KUKA KRL program: EPS_2_251349_CBMH082_A_20251001124258.src

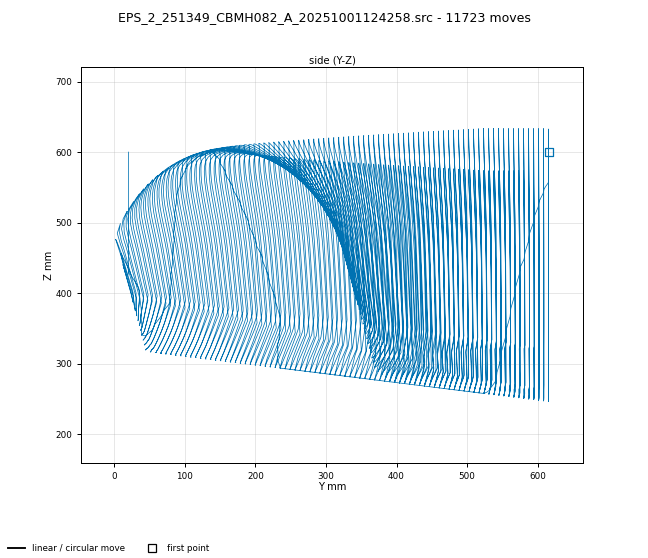
[picture p0: tool path of EPS_2_251349_CBMH082_A_20251001124258.src, 11723 of 11725 moves have a stored position in this frame; points joined in program order, loops and branches not executed]
&ACCESS RVP
&REL 4
&COMMENT QRS 19112012
&PARAM EDITMASK = *
DEF PART()
EXT BAS (BAS_COMMAND :IN,REAL :IN )
INT I
BAS (#INITMOV,0 )

;KUKA QRS Post kuka4.cps  Date:22-06-2017 !

File_ID=2859

QRS_PRE_INIT()

;Init var - Until changes are made in qrs_pre_init
Outlet_Square_prg=0
Inlet_1_Square_prg=0
Inlet_2_Square_prg=0
Inlet_3_Square_prg=0
Inlet_4_Square_prg=0
Inlet_5_Square_prg=0

Outlet_1={X 0.000, Y 523.550, Z 484.000, B 0.000, E1 0.000 }
Inlet_1={X 0.000, Y 527.930, Z 424.000, B 0.000, E1 90.000 }
Outlet_1_type=299
Inlet_1_type=299
;QRS#1=Sidecore dimensions
;QRS#2=300-12" PVC SDR 35
;QRS#3=300-12" PVC SDR 35
;QRS#4=
;QRS#5=
;QRS#6=
;QRS#7=
;QRS#8=
;QRS#9=16M PSX
;QRS#10=16M PSX
;QRS#11=
;QRS#12=
;QRS#13=
;QRS#14=
;QRS#15=
;QRS#16=1220x127x914 3'
;QRS#17=EPS Height
;QRS#18=633,5
;QRS#19=*
;QRS#20= UPDATED VERSION 22-06-2017
;QRS#21=*
Outlet_Square=0150
Inlet_1_Square=0150
Inlet_2_Square=0
Inlet_3_Square=0
Inlet_4_Square=0
Inlet_5_Square=0
Mill_Square=1
Outlet_Square_Prg=206
Inlet_1_Square_prg=206

QRS_INIT()

$ADVANCE=5

; T1
PTP {E1 173.526,E2 173.526}
PTP {X 0,Y 615.503,A -85,B 0,C 180,E1 173.526,E2 173.526,E3 0,E4 0,E5 0,E6 0}
QRS_SPEED_INIT()
LIN {X 0,Y 615.503,Z 600,A -85,B 0,C 180,E1 173.526,E2 173.526,E3 0,E4 0,E5 0,E6 0} C_VEL
LIN {X 0,Y 615.503,Z 569.829,A -85,B 0,C 180,E1 173.526,E2 173.526} C_VEL
LIN {X 0,Y 615.503,Z 560.181,A -85,B 0,C 180,E1 173.526,E2 173.526} C_VEL
LIN {X 0,Y 615.497,Z 558.359,A -85,B 0,C 180,E1 173.417,E2 173.417} C_VEL
LIN {X 0,Y 615.491,Z 551.664,A -85,B 0,C 180,E1 172.125,E2 172.125} C_VEL
LIN {X 0,Y 615.491,Z 543.149,A -85,B 0,C 180,E1 170.802,E2 170.802} C_VEL
LIN {X 0,Y 615.497,Z 534.071,A -85,B 0,C 180,E1 169.64,E2 169.64} C_VEL
LIN {X 0,Y 615.492,Z 524.798,A -85,B 0,C 180,E1 168.641,E2 168.641} C_VEL
LIN {X 0,Y 615.497,Z 512.83,A -85,B 0,C 180,E1 167.554,E2 167.554} C_VEL
LIN {X 0,Y 615.497,Z 500.591,A -85,B 0,C 180,E1 166.632,E2 166.632} C_VEL
LIN {X 0,Y 615.499,Z 487.891,A -85,B 0,C 180,E1 165.835,E2 165.835} C_VEL
LIN {X 0,Y 615.49,Z 473.795,A -85,B 0,C 180,E1 165.113,E2 165.113} C_VEL
LIN {X 0,Y 615.495,Z 459.141,A -85,B 0,C 180,E1 164.52,E2 164.52} C_VEL
LIN {X 0,Y 615.491,Z 444.202,A -85,B 0,C 180,E1 164.063,E2 164.063} C_VEL
LIN {X 0,Y 615.486,Z 428.985,A -85,B 0,C 180,E1 163.738,E2 163.738} C_VEL
LIN {X 0,Y 615.463,Z 380.474,A -85,B 0,C 180,E1 163.136,E2 163.136} C_VEL
LIN {X 0,Y 615.477,Z 263.406,A -85,B 0,C 180,E1 161.724,E2 161.724} C_VEL
LIN {X 0,Y 615.454,Z 246.316,A -85,B 0,C 180,E1 159.315,E2 159.315} C_VEL
LIN {X 0,Y 615.493,Z 246.313,A -85,B 0,C 180,E1 156.445,E2 156.445} C_VEL
LIN {X 0,Y 615.457,Z 246.319,A -85,B 0,C 180,E1 153.555,E2 153.555} C_VEL
LIN {X 0,Y 615.454,Z 246.316,A -85,B 0,C 180,E1 151.341,E2 151.341} C_VEL
LIN {X 0,Y 615.474,Z 246.311,A -85,B 0,C 180,E1 148.917,E2 148.917} C_VEL
LIN {X 0,Y 615.481,Z 246.324,A -85,B 0,C 180,E1 145.979,E2 145.979} C_VEL
LIN {X 0,Y 615.456,Z 246.318,A -85,B 0,C 180,E1 143.574,E2 143.574} C_VEL
LIN {X 0,Y 615.473,Z 246.311,A -85,B 0,C 180,E1 140.94,E2 140.94} C_VEL
LIN {X 0,Y 615.474,Z 246.322,A -85,B 0,C 180,E1 137.922,E2 137.922} C_VEL
LIN {X 0,Y 615.467,Z 246.321,A -85,B 0,C 180,E1 135.85,E2 135.85} C_VEL
LIN {X 0,Y 615.458,Z 246.314,A -85,B 0,C 180,E1 133.248,E2 133.248} C_VEL
LIN {X 0,Y 615.488,Z 246.314,A -85,B 0,C 180,E1 130.607,E2 130.607} C_VEL
LIN {X 0,Y 615.477,Z 246.323,A -85,B 0,C 180,E1 128.012,E2 128.012} C_VEL
LIN {X 0,Y 615.453,Z 246.318,A -85,B 0,C 180,E1 125.619,E2 125.619} C_VEL
LIN {X 0,Y 615.461,Z 246.313,A -85,B 0,C 180,E1 123.239,E2 123.239} C_VEL
LIN {X 0,Y 615.489,Z 246.309,A -85,B 0,C 180,E1 120.92,E2 120.92} C_VEL
LIN {X 0,Y 615.464,Z 246.321,A -85,B 0,C 180,E1 117.917,E2 117.917} C_VEL
LIN {X 0,Y 615.452,Z 246.317,A -85,B 0,C 180,E1 115.564,E2 115.564} C_VEL
LIN {X 0,Y 615.487,Z 246.312,A -85,B 0,C 180,E1 112.845,E2 112.845} C_VEL
LIN {X 0,Y 615.469,Z 246.322,A -85,B 0,C 180,E1 110.034,E2 110.034} C_VEL
LIN {X 0,Y 615.463,Z 246.321,A -85,B 0,C 180,E1 107.958,E2 107.958} C_VEL
LIN {X 0,Y 615.459,Z 246.32,A -85,B 0,C 180,E1 105.907,E2 105.907} C_VEL
LIN {X 0,Y 615.457,Z 246.319,A -85,B 0,C 180,E1 103.876,E2 103.876} C_VEL
LIN {X 0,Y 615.472,Z 246.311,A -85,B 0,C 180,E1 101.194,E2 101.194} C_VEL
LIN {X 0,Y 615.491,Z 246.322,A -85,B 0,C 180,E1 98.537,E2 98.537} C_VEL
LIN {X 0,Y 615.456,Z 246.319,A -85,B 0,C 180,E1 95.9,E2 95.9} C_VEL
LIN {X 0,Y 615.469,Z 246.312,A -85,B 0,C 180,E1 93.274,E2 93.274} C_VEL
LIN {X 0,Y 615.493,Z 246.319,A -85,B 0,C 180,E1 90.655,E2 90.655} C_VEL
LIN {X 0,Y 615.461,Z 246.32,A -85,B 0,C 180,E1 88.038,E2 88.038} C_VEL
LIN {X 0,Y 615.461,Z 246.313,A -85,B 0,C 180,E1 85.416,E2 85.416} C_VEL
LIN {X 0,Y 615.493,Z 246.316,A -85,B 0,C 180,E1 82.785,E2 82.785} C_VEL
LIN {X 0,Y 615.464,Z 246.321,A -85,B 0,C 180,E1 80.138,E2 80.138} C_VEL
LIN {X 0,Y 615.461,Z 246.313,A -85,B 0,C 180,E1 77.47,E2 77.47} C_VEL
LIN {X 0,Y 615.493,Z 246.318,A -85,B 0,C 180,E1 74.775,E2 74.775} C_VEL
LIN {X 0,Y 615.456,Z 246.319,A -85,B 0,C 180,E1 72.043,E2 72.043} C_VEL
LIN {X 0,Y 615.466,Z 246.312,A -85,B 0,C 180,E1 69.446,E2 69.446} C_VEL
LIN {X 0,Y 615.485,Z 246.311,A -85,B 0,C 180,E1 67.157,E2 67.157} C_VEL
LIN {X 0,Y 615.464,Z 246.322,A -85,B 0,C 180,E1 64.285,E2 64.285} C_VEL
LIN {X 0,Y 615.454,Z 246.319,A -85,B 0,C 180,E1 62.085,E2 62.085} C_VEL
LIN {X 0,Y 615.449,Z 246.317,A -85,B 0,C 180,E1 59.839,E2 59.839} C_VEL
LIN {X 0,Y 615.464,Z 246.313,A -85,B 0,C 180,E1 57.543,E2 57.543} C_VEL
LIN {X 0,Y 615.499,Z 246.309,A -85,B 0,C 180,E1 55.187,E2 55.187} C_VEL
LIN {X 0,Y 615.488,Z 246.324,A -85,B 0,C 180,E1 52.759,E2 52.759} C_VEL
LIN {X 0,Y 615.459,Z 246.32,A -85,B 0,C 180,E1 50.249,E2 50.249} C_VEL
LIN {X 0,Y 615.457,Z 246.314,A -85,B 0,C 180,E1 47.646,E2 47.646} C_VEL
LIN {X 0,Y 615.489,Z 246.319,A -85,B 0,C 180,E1 44.933,E2 44.933} C_VEL
LIN {X 0,Y 615.463,Z 246.321,A -85,B 0,C 180,E1 42.354,E2 42.354} C_VEL
LIN {X 0,Y 615.457,Z 246.314,A -85,B 0,C 180,E1 39.751,E2 39.751} C_VEL
LIN {X 0,Y 615.486,Z 246.322,A -85,B 0,C 180,E1 36.939,E2 36.939} C_VEL
LIN {X 0,Y 615.448,Z 246.317,A -85,B 0,C 180,E1 34.023,E2 34.023} C_VEL
LIN {X 0,Y 615.494,Z 246.316,A -85,B 0,C 180,E1 31.09,E2 31.09} C_VEL
LIN {X 0,Y 615.463,Z 246.321,A -85,B 0,C 180,E1 28.449,E2 28.449} C_VEL
LIN {X 0,Y 615.462,Z 246.321,A -85,B 0,C 180,E1 26.444,E2 26.444} C_VEL
LIN {X 0,Y 615.449,Z 246.316,A -85,B 0,C 180,E1 24.004,E2 24.004} C_VEL
LIN {X 0,Y 615.492,Z 246.31,A -85,B 0,C 180,E1 21.431,E2 21.431} C_VEL
LIN {X 0,Y 615.47,Z 246.322,A -85,B 0,C 180,E1 18.604,E2 18.604} C_VEL
LIN {X 0,Y 615.457,Z 246.32,A -85,B 0,C 180,E1 16.427,E2 16.427} C_VEL
LIN {X 0,Y 615.458,Z 246.314,A -85,B 0,C 180,E1 13.874,E2 13.874} C_VEL
LIN {X 0,Y 615.485,Z 246.328,A -85,B 0,C 180,E1 10.895,E2 10.895} C_VEL
LIN {X 0,Y 615.461,Z 246.321,A -85,B 0,C 180,E1 8.536,E2 8.536} C_VEL
LIN {X 0,Y 615.459,Z 246.314,A -85,B 0,C 180,E1 5.898,E2 5.898} C_VEL
LIN {X 0,Y 615.494,Z 246.316,A -85,B 0,C 180,E1 3.272,E2 3.272} C_VEL
LIN {X 0,Y 615.466,Z 246.322,A -85,B 0,C 180,E1 0.654,E2 0.654} C_VEL
LIN {X 0,Y 615.454,Z 246.315,A -85,B 0,C 180,E1 -1.964,E2 -1.964} C_VEL
LIN {X 0,Y 615.496,Z 246.313,A -85,B 0,C 180,E1 -4.585,E2 -4.585} C_VEL
LIN {X 0,Y 615.473,Z 246.322,A -85,B 0,C 180,E1 -7.216,E2 -7.216} C_VEL
LIN {X 0,Y 615.45,Z 246.316,A -85,B 0,C 180,E1 -9.863,E2 -9.863} C_VEL
LIN {X 0,Y 615.49,Z 246.314,A -85,B 0,C 180,E1 -12.53,E2 -12.53} C_VEL
LIN {X 0,Y 615.468,Z 246.322,A -85,B 0,C 180,E1 -15.227,E2 -15.227} C_VEL
LIN {X 0,Y 615.463,Z 246.321,A -85,B 0,C 180,E1 -17.272,E2 -17.272} C_VEL
LIN {X 0,Y 615.454,Z 246.321,A -85,B 0,C 180,E1 -19.339,E2 -19.339} C_VEL
LIN {X 0,Y 615.453,Z 246.319,A -85,B 0,C 180,E1 -21.433,E2 -21.433} C_VEL
LIN {X 0,Y 615.459,Z 246.314,A -85,B 0,C 180,E1 -24.006,E2 -24.006} C_VEL
LIN {X 0,Y 615.497,Z 246.312,A -85,B 0,C 180,E1 -26.444,E2 -26.444} C_VEL
LIN {X 0,Y 615.494,Z 246.319,A -85,B 0,C 180,E1 -28.658,E2 -28.658} C_VEL
LIN {X 0,Y 615.471,Z 246.322,A -85,B 0,C 180,E1 -31.086,E2 -31.086} C_VEL
LIN {X 0,Y 615.449,Z 246.318,A -85,B 0,C 180,E1 -33.531,E2 -33.531} C_VEL
LIN {X 0,Y 615.455,Z 246.314,A -85,B 0,C 180,E1 -35.832,E2 -35.832} C_VEL
LIN {X 0,Y 615.475,Z 246.312,A -85,B 0,C 180,E1 -38.07,E2 -38.07} C_VEL
LIN {X 0,Y 615.466,Z 246.322,A -85,B 0,C 180,E1 -41.094,E2 -41.094} C_VEL
LIN {X 0,Y 615.455,Z 246.32,A -85,B 0,C 180,E1 -43.248,E2 -43.248} C_VEL
LIN {X 0,Y 615.472,Z 246.312,A -85,B 0,C 180,E1 -46.004,E2 -46.004} C_VEL
LIN {X 0,Y 615.476,Z 246.324,A -85,B 0,C 180,E1 -48.907,E2 -48.907} C_VEL
LIN {X 0,Y 615.461,Z 246.321,A -85,B 0,C 180,E1 -51.095,E2 -51.095} C_VEL
LIN {X 0,Y 615.45,Z 246.316,A -85,B 0,C 180,E1 -53.574,E2 -53.574} C_VEL
LIN {X 0,Y 615.494,Z 246.318,A -85,B 0,C 180,E1 -56.465,E2 -56.465} C_VEL
LIN {X 0,Y 615.457,Z 246.321,A -85,B 0,C 180,E1 -59.08,E2 -59.08} C_VEL
LIN {X 0,Y 615.45,Z 246.316,A -85,B 0,C 180,E1 -61.556,E2 -61.556} C_VEL
LIN {X 0,Y 615.462,Z 246.374,A -85,B 0,C 180,E1 -63.784,E2 -63.784} C_VEL
LIN {X 0,Y 615.485,Z 272.614,A -85,B 0,C 180,E1 -66.623,E2 -66.623} C_VEL
LIN {X 0,Y 615.486,Z 299.254,A -85,B 0,C 180,E1 -69.443,E2 -69.443} C_VEL
LIN {X 0,Y 615.495,Z 321.324,A -85,B 0,C 180,E1 -71.741,E2 -71.741} C_VEL
LIN {X 0,Y 615.487,Z 488.149,A -85,B 0,C 180,E1 -73.768,E2 -73.768} C_VEL
LIN {X 0,Y 615.49,Z 503.756,A -85,B 0,C 180,E1 -74.096,E2 -74.096} C_VEL
LIN {X 0,Y 615.48,Z 519.082,A -85,B 0,C 180,E1 -74.563,E2 -74.563} C_VEL
LIN {X 0,Y 615.492,Z 532.779,A -85,B 0,C 180,E1 -75.114,E2 -75.114} C_VEL
LIN {X 0,Y 615.494,Z 547.055,A -85,B 0,C 180,E1 -75.834,E2 -75.834} C_VEL
LIN {X 0,Y 615.497,Z 559.915,A -85,B 0,C 180,E1 -76.632,E2 -76.632} C_VEL
LIN {X 0,Y 615.495,Z 572.268,A -85,B 0,C 180,E1 -77.555,E2 -77.555} C_VEL
LIN {X 0,Y 615.495,Z 582.618,A -85,B 0,C 180,E1 -78.474,E2 -78.474} C_VEL
LIN {X 0,Y 615.495,Z 592.193,A -85,B 0,C 180,E1 -79.474,E2 -79.474} C_VEL
LIN {X 0,Y 615.494,Z 601.585,A -85,B 0,C 180,E1 -80.637,E2 -80.637} C_VEL
LIN {X 0,Y 615.495,Z 609.387,A -85,B 0,C 180,E1 -81.795,E2 -81.795} C_VEL
LIN {X 0,Y 615.496,Z 616.609,A -85,B 0,C 180,E1 -83.102,E2 -83.102} C_VEL
LIN {X 0,Y 615.499,Z 622.44,A -85,B 0,C 180,E1 -84.431,E2 -84.431} C_VEL
LIN {X 0,Y 615.491,Z 625.863,A -85,B 0,C 180,E1 -85.416,E2 -85.416} C_VEL
LIN {X 0,Y 615.492,Z 629.32,A -85,B 0,C 180,E1 -86.728,E2 -86.728} C_VEL
LIN {X 0,Y 615.497,Z 631.594,A -85,B 0,C 180,E1 -88.038,E2 -88.038} C_VEL
LIN {X 0,Y 615.493,Z 632.741,A -85,B 0,C 180,E1 -89.347,E2 -89.347} C_VEL
LIN {X 0,Y 615.493,Z 632.74,A -85,B 0,C 180,E1 -90.655,E2 -90.655} C_VEL
LIN {X 0,Y 615.497,Z 631.592,A -85,B 0,C 180,E1 -91.964,E2 -91.964} C_VEL
LIN {X 0,Y 615.492,Z 629.316,A -85,B 0,C 180,E1 -93.274,E2 -93.274} C_VEL
LIN {X 0,Y 615.491,Z 625.857,A -85,B 0,C 180,E1 -94.585,E2 -94.585} C_VEL
LIN {X 0,Y 615.49,Z 621.14,A -85,B 0,C 180,E1 -95.899,E2 -95.899} C_VEL
LIN {X 0,Y 615.495,Z 615.025,A -85,B 0,C 180,E1 -97.216,E2 -97.216} C_VEL
LIN {X 0,Y 615.49,Z 607.327,A -85,B 0,C 180,E1 -98.537,E2 -98.537} C_VEL
LIN {X 0,Y 615.495,Z 599.107,A -85,B 0,C 180,E1 -99.697,E2 -99.697} C_VEL
LIN {X 0,Y 615.497,Z 588.896,A -85,B 0,C 180,E1 -100.892,E2 -100.892} C_VEL
LIN {X 0,Y 615.495,Z 579.059,A -85,B 0,C 180,E1 -101.861,E2 -101.861} C_VEL
LIN {X 0,Y 615.498,Z 566.936,A -85,B 0,C 180,E1 -102.866,E2 -102.866} C_VEL
LIN {X 0,Y 615.498,Z 554.785,A -85,B 0,C 180,E1 -103.706,E2 -103.706} C_VEL
LIN {X 0,Y 615.484,Z 541.367,A -85,B 0,C 180,E1 -104.473,E2 -104.473} C_VEL
LIN {X 0,Y 615.495,Z 526.83,A -85,B 0,C 180,E1 -105.142,E2 -105.142} C_VEL
LIN {X 0,Y 615.484,Z 512.592,A -85,B 0,C 180,E1 -105.651,E2 -105.651} C_VEL
LIN {X 0,Y 615.499,Z 498.103,A -85,B 0,C 180,E1 -106.036,E2 -106.036} C_VEL
LIN {X 0,Y 615.487,Z 483.529,A -85,B 0,C 180,E1 -106.298,E2 -106.298} C_VEL
LIN {X 0,Y 615.494,Z 321.314,A -85,B 0,C 180,E1 -108.26,E2 -108.26} C_VEL
LIN {X 0,Y 615.484,Z 295.921,A -85,B 0,C 180,E1 -110.907,E2 -110.907} C_VEL
LIN {X 0,Y 615.491,Z 268.818,A -85,B 0,C 180,E1 -113.783,E2 -113.783} C_VEL
LIN {X 0,Y 615.463,Z 246.356,A -85,B 0,C 180,E1 -116.218,E2 -116.218} C_VEL
LIN {X 0,Y 615.455,Z 246.318,A -85,B 0,C 180,E1 -118.66,E2 -118.66} C_VEL
LIN {X 0,Y 615.485,Z 246.324,A -85,B 0,C 180,E1 -121.085,E2 -121.085} C_VEL
LIN {X 0,Y 615.478,Z 246.31,A -85,B 0,C 180,E1 -124.023,E2 -124.023} C_VEL
LIN {X 0,Y 615.464,Z 246.316,A -85,B 0,C 180,E1 -126.427,E2 -126.427} C_VEL
LIN {X 0,Y 615.493,Z 246.324,A -85,B 0,C 180,E1 -129.063,E2 -129.063} C_VEL
LIN {X 0,Y 615.484,Z 246.313,A -85,B 0,C 180,E1 -131.475,E2 -131.475} C_VEL
LIN {X 0,Y 615.475,Z 246.313,A -85,B 0,C 180,E1 -134.151,E2 -134.151} C_VEL
LIN {X 0,Y 615.486,Z 246.321,A -85,B 0,C 180,E1 -136.953,E2 -136.953} C_VEL
LIN {X 0,Y 615.479,Z 246.312,A -85,B 0,C 180,E1 -139.393,E2 -139.393} C_VEL
LIN {X 0,Y 615.484,Z 246.311,A -85,B 0,C 180,E1 -141.989,E2 -141.989} C_VEL
LIN {X 0,Y 615.489,Z 246.321,A -85,B 0,C 180,E1 -144.384,E2 -144.384} C_VEL
LIN {X 0,Y 615.476,Z 246.321,A -85,B 0,C 180,E1 -146.763,E2 -146.763} C_VEL
LIN {X 0,Y 615.465,Z 246.315,A -85,B 0,C 180,E1 -149.079,E2 -149.079} C_VEL
LIN {X 0,Y 615.489,Z 246.308,A -85,B 0,C 180,E1 -151.55,E2 -151.55} C_VEL
LIN {X 0,Y 615.483,Z 246.323,A -85,B 0,C 180,E1 -154.433,E2 -154.433} C_VEL
LIN {X 0,Y 615.46,Z 246.314,A -85,B 0,C 180,E1 -157.154,E2 -157.154} C_VEL
LIN {X 0,Y 615.48,Z 246.437,A -85,B 0,C 180,E1 -159.446,E2 -159.446} C_VEL
LIN {X 0,Y 615.494,Z 263.458,A -85,B 0,C 180,E1 -161.822,E2 -161.822} C_VEL
LIN {X 0,Y 615.497,Z 427.262,A -85,B 0,C 180,E1 -163.8,E2 -163.8} C_VEL
LIN {X 0,Y 615.494,Z 441.803,A -85,B 0,C 180,E1 -164.095,E2 -164.095} C_VEL
LIN {X 0,Y 615.496,Z 456.406,A -85,B 0,C 180,E1 -164.519,E2 -164.519} C_VEL
LIN {X 0,Y 615.489,Z 469.73,A -85,B 0,C 180,E1 -165.028,E2 -165.028} C_VEL
LIN {X 0,Y 615.493,Z 483.381,A -85,B 0,C 180,E1 -165.681,E2 -165.681} C_VEL
LIN {X 0,Y 615.5,Z 496.661,A -85,B 0,C 180,E1 -166.462,E2 -166.462} C_VEL
LIN {X 0,Y 615.497,Z 508.512,A -85,B 0,C 180,E1 -167.302,E2 -167.302} C_VEL
LIN {X 0,Y 615.497,Z 520.356,A -85,B 0,C 180,E1 -168.306,E2 -168.306} C_VEL
LIN {X 0,Y 615.495,Z 530.169,A -85,B 0,C 180,E1 -169.292,E2 -169.292} C_VEL
LIN {X 0,Y 615.498,Z 540.009,A -85,B 0,C 180,E1 -170.469,E2 -170.469} C_VEL
LIN {X 0,Y 615.496,Z 548.1,A -85,B 0,C 180,E1 -171.628,E2 -171.628} C_VEL
LIN {X 0,Y 615.493,Z 554.78,A -85,B 0,C 180,E1 -172.784,E2 -172.784} C_VEL
LIN {X 0,Y 615.488,Z 560.948,A -85,B 0,C 180,E1 -174.101,E2 -174.101} C_VEL
LIN {X 0,Y 615.489,Z 565.715,A -85,B 0,C 180,E1 -175.415,E2 -175.415} C_VEL
LIN {X 0,Y 615.496,Z 569.219,A -85,B 0,C 180,E1 -176.727,E2 -176.727} C_VEL
LIN {X 0,Y 615.493,Z 571.541,A -85,B 0,C 180,E1 -178.036,E2 -178.036} C_VEL
LIN {X 0,Y 615.491,Z 572.728,A -85,B 0,C 180,E1 -179.345,E2 -179.345} C_VEL
LIN {X 0,Y 615.494,Z 572.751,A -85,B 0,C 180,E1 -180.654,E2 -180.654} C_VEL
LIN {X 0,Y 615.497,Z 571.647,A -85,B 0,C 180,E1 -181.963,E2 -181.963} C_VEL
LIN {X 0,Y 615.497,Z 569.416,A -85,B 0,C 180,E1 -183.272,E2 -183.272} C_VEL
LIN {X 0,Y 615.496,Z 566.005,A -85,B 0,C 180,E1 -184.584,E2 -184.584} C_VEL
LIN {X 0,Y 615.49,Z 561.34,A -85,B 0,C 180,E1 -185.898,E2 -185.898} C_VEL
LIN {X 0,Y 615.497,Z 558.359,A -85,B 0,C 180,E1 -186.583,E2 -186.583} C_VEL
LIN {X 0,Y 614.828,Z 556.102,A -85,B 0,C 180,E1 -187.082,E2 -187.082} C_VEL
LIN {X 0,Y 612.006,Z 552.209,A -85,B 0,C 180,E1 -187.888,E2 -187.888} C_VEL
LIN {X 0,Y 609.154,Z 547.637,A -85,B 0,C 180,E1 -188.679,E2 -188.679} C_VEL
LIN {X 0,Y 608.464,Z 544.491,A -85,B 0,C 180,E1 -189.153,E2 -189.153} C_VEL
LIN {X 0,Y 608.478,Z 535.67,A -85,B 0,C 180,E1 -190.312,E2 -190.312} C_VEL
LIN {X 0,Y 608.494,Z 524.953,A -85,B 0,C 180,E1 -191.492,E2 -191.492} C_VEL
LIN {X 0,Y 608.513,Z 512.908,A -85,B 0,C 180,E1 -192.591,E2 -192.591} C_VEL
LIN {X 0,Y 608.543,Z 500.629,A -85,B 0,C 180,E1 -193.524,E2 -193.524} C_VEL
LIN {X 0,Y 608.577,Z 487.683,A -85,B 0,C 180,E1 -194.341,E2 -194.341} C_VEL
LIN {X 0,Y 608.605,Z 473.771,A -85,B 0,C 180,E1 -195.059,E2 -195.059} C_VEL
LIN {X 0,Y 608.639,Z 459.125,A -85,B 0,C 180,E1 -195.658,E2 -195.658} C_VEL
LIN {X 0,Y 608.661,Z 443.559,A -85,B 0,C 180,E1 -196.137,E2 -196.137} C_VEL
LIN {X 0,Y 608.678,Z 427.766,A -85,B 0,C 180,E1 -196.469,E2 -196.469} C_VEL
LIN {X 0,Y 608.638,Z 264.297,A -85,B 0,C 180,E1 -198.468,E2 -198.468} C_VEL
LIN {X 0,Y 608.509,Z 263.438,A -85,B 0,C 180,E1 -198.492,E2 -198.492} C_VEL
LIN {X 0,Y 608.466,Z 247.558,A -85,B 0,C 180,E1 -200.735,E2 -200.735} C_VEL
LIN {X 0,Y 608.444,Z 247.315,A -85,B 0,C 180,E1 -200.981,E2 -200.981} C_VEL
LIN {X 0,Y 608.469,Z 247.319,A -85,B 0,C 180,E1 -203.844,E2 -203.844} C_VEL
LIN {X 0,Y 608.437,Z 247.323,A -85,B 0,C 180,E1 -206.035,E2 -206.035} C_VEL
LIN {X 0,Y 608.447,Z 247.314,A -85,B 0,C 180,E1 -208.615,E2 -208.615} C_VEL
LIN {X 0,Y 608.445,Z 247.315,A -85,B 0,C 180,E1 -211.317,E2 -211.317} C_VEL
LIN {X 0,Y 608.475,Z 247.317,A -85,B 0,C 180,E1 -213.735,E2 -213.735} C_VEL
LIN {X 0,Y 608.442,Z 247.32,A -85,B 0,C 180,E1 -216.091,E2 -216.091} C_VEL
LIN {X 0,Y 608.424,Z 247.316,A -85,B 0,C 180,E1 -218.59,E2 -218.59} C_VEL
LIN {X 0,Y 608.461,Z 247.314,A -85,B 0,C 180,E1 -221.341,E2 -221.341} C_VEL
LIN {X 0,Y 608.465,Z 247.321,A -85,B 0,C 180,E1 -223.869,E2 -223.869} C_VEL
LIN {X 0,Y 608.449,Z 247.313,A -85,B 0,C 180,E1 -226.692,E2 -226.692} C_VEL
LIN {X 0,Y 608.434,Z 247.314,A -85,B 0,C 180,E1 -228.821,E2 -228.821} C_VEL
LIN {X 0,Y 608.464,Z 247.322,A -85,B 0,C 180,E1 -231.759,E2 -231.759} C_VEL
LIN {X 0,Y 608.439,Z 247.321,A -85,B 0,C 180,E1 -233.954,E2 -233.954} C_VEL
LIN {X 0,Y 608.437,Z 247.316,A -85,B 0,C 180,E1 -236.327,E2 -236.327} C_VEL
LIN {X 0,Y 608.437,Z 247.314,A -85,B 0,C 180,E1 -238.732,E2 -238.732} C_VEL
LIN {X 0,Y 608.478,Z 247.314,A -85,B 0,C 180,E1 -241.377,E2 -241.377} C_VEL
LIN {X 0,Y 608.444,Z 247.315,A -85,B 0,C 180,E1 -244.282,E2 -244.282} C_VEL
LIN {X 0,Y 608.439,Z 247.314,A -85,B 0,C 180,E1 -246.875,E2 -246.875} C_VEL
LIN {X 0,Y 608.457,Z 247.322,A -85,B 0,C 180,E1 -249.725,E2 -249.725} C_VEL
LIN {X 0,Y 608.435,Z 247.322,A -85,B 0,C 180,E1 -251.827,E2 -251.827} C_VEL
LIN {X 0,Y 608.448,Z 247.319,A -85,B 0,C 180,E1 -253.905,E2 -253.905} C_VEL
LIN {X 0,Y 608.445,Z 247.318,A -85,B 0,C 180,E1 -255.988,E2 -255.988} C_VEL
LIN {X 0,Y 608.446,Z 247.313,A -85,B 0,C 180,E1 -258.675,E2 -258.675} C_VEL
LIN {X 0,Y 608.457,Z 247.318,A -85,B 0,C 180,E1 -261.363,E2 -261.363} C_VEL
LIN {X 0,Y 608.435,Z 247.318,A -85,B 0,C 180,E1 -264.032,E2 -264.032} C_VEL
LIN {X 0,Y 608.462,Z 247.311,A -85,B 0,C 180,E1 -266.688,E2 -266.688} C_VEL
LIN {X 0,Y 608.486,Z 247.315,A -85,B 0,C 180,E1 -269.337,E2 -269.337} C_VEL
LIN {X 0,Y 608.431,Z 247.318,A -85,B 0,C 180,E1 -271.985,E2 -271.985} C_VEL
LIN {X 0,Y 608.43,Z 247.318,A -85,B 0,C 180,E1 -273.973,E2 -273.973} C_VEL
LIN {X 0,Y 608.449,Z 247.313,A -85,B 0,C 180,E1 -276.632,E2 -276.632} C_VEL
LIN {X 0,Y 608.469,Z 247.317,A -85,B 0,C 180,E1 -279.305,E2 -279.305} C_VEL
LIN {X 0,Y 608.44,Z 247.316,A -85,B 0,C 180,E1 -281.999,E2 -281.999} C_VEL
LIN {X 0,Y 608.461,Z 247.312,A -85,B 0,C 180,E1 -284.72,E2 -284.72} C_VEL
LIN {X 0,Y 608.448,Z 247.324,A -85,B 0,C 180,E1 -287.476,E2 -287.476} C_VEL
LIN {X 0,Y 608.437,Z 247.314,A -85,B 0,C 180,E1 -290.274,E2 -290.274} C_VEL
LIN {X 0,Y 608.445,Z 247.313,A -85,B 0,C 180,E1 -292.476,E2 -292.476} C_VEL
LIN {X 0,Y 608.449,Z 247.322,A -85,B 0,C 180,E1 -295.3,E2 -295.3} C_VEL
LIN {X 0,Y 608.437,Z 247.323,A -85,B 0,C 180,E1 -297.517,E2 -297.517} C_VEL
LIN {X 0,Y 608.438,Z 247.316,A -85,B 0,C 180,E1 -299.969,E2 -299.969} C_VEL
LIN {X 0,Y 608.441,Z 247.314,A -85,B 0,C 180,E1 -302.521,E2 -302.521} C_VEL
LIN {X 0,Y 608.44,Z 247.323,A -85,B 0,C 180,E1 -305.276,E2 -305.276} C_VEL
LIN {X 0,Y 608.447,Z 247.317,A -85,B 0,C 180,E1 -307.746,E2 -307.746} C_VEL
LIN {X 0,Y 608.427,Z 247.315,A -85,B 0,C 180,E1 -310.328,E2 -310.328} C_VEL
LIN {X 0,Y 608.455,Z 247.317,A -85,B 0,C 180,E1 -312.958,E2 -312.958} C_VEL
LIN {X 0,Y 608.427,Z 247.319,A -85,B 0,C 180,E1 -315.737,E2 -315.737} C_VEL
LIN {X 0,Y 608.432,Z 247.316,A -85,B 0,C 180,E1 -317.937,E2 -317.937} C_VEL
LIN {X 0,Y 608.467,Z 247.313,A -85,B 0,C 180,E1 -320.701,E2 -320.701} C_VEL
LIN {X 0,Y 608.455,Z 247.32,A -85,B 0,C 180,E1 -323.086,E2 -323.086} C_VEL
LIN {X 0,Y 608.458,Z 247.317,A -85,B 0,C 180,E1 -325.531,E2 -325.531} C_VEL
LIN {X 0,Y 608.441,Z 247.315,A -85,B 0,C 180,E1 -327.905,E2 -327.905} C_VEL
LIN {X 0,Y 608.443,Z 247.313,A -85,B 0,C 180,E1 -330.22,E2 -330.22} C_VEL
LIN {X 0,Y 608.479,Z 247.313,A -85,B 0,C 180,E1 -332.789,E2 -332.789} C_VEL
LIN {X 0,Y 608.437,Z 247.32,A -85,B 0,C 180,E1 -335.429,E2 -335.429} C_VEL
LIN {X 0,Y 608.458,Z 247.312,A -85,B 0,C 180,E1 -338.309,E2 -338.309} C_VEL
LIN {X 0,Y 608.456,Z 247.32,A -85,B 0,C 180,E1 -341.284,E2 -341.284} C_VEL
LIN {X 0,Y 608.431,Z 247.315,A -85,B 0,C 180,E1 -343.906,E2 -343.906} C_VEL
LIN {X 0,Y 608.462,Z 247.314,A -85,B 0,C 180,E1 -346.644,E2 -346.644} C_VEL
LIN {X 0,Y 608.448,Z 247.319,A -85,B 0,C 180,E1 -349.351,E2 -349.351} C_VEL
LIN {X 0,Y 608.453,Z 247.312,A -85,B 0,C 180,E1 -352.033,E2 -352.033} C_VEL
LIN {X 0,Y 608.469,Z 247.315,A -85,B 0,C 180,E1 -354.699,E2 -354.699} C_VEL
LIN {X 0,Y 608.457,Z 247.317,A -85,B 0,C 180,E1 -357.352,E2 -357.352} C_VEL
LIN {X 0,Y 608.448,Z 247.313,A -85,B 0,C 180,E1 -360.001,E2 -360.001} C_VEL
LIN {X 0,Y 608.483,Z 247.313,A -85,B 0,C 180,E1 -362.649,E2 -362.649} C_VEL
LIN {X 0,Y 608.449,Z 247.318,A -85,B 0,C 180,E1 -365.302,E2 -365.302} C_VEL
LIN {X 0,Y 608.451,Z 247.312,A -85,B 0,C 180,E1 -367.968,E2 -367.968} C_VEL
LIN {X 0,Y 608.468,Z 247.321,A -85,B 0,C 180,E1 -370.963,E2 -370.963} C_VEL
LIN {X 0,Y 608.442,Z 247.317,A -85,B 0,C 180,E1 -373.357,E2 -373.357} C_VEL
LIN {X 0,Y 608.45,Z 247.316,A -85,B 0,C 180,E1 -375.407,E2 -375.407} C_VEL
LIN {X 0,Y 608.429,Z 247.317,A -85,B 0,C 180,E1 -377.478,E2 -377.478} C_VEL
LIN {X 0,Y 608.425,Z 247.317,A -85,B 0,C 180,E1 -379.572,E2 -379.572} C_VEL
LIN {X 0,Y 608.443,Z 247.314,A -85,B 0,C 180,E1 -381.693,E2 -381.693} C_VEL
LIN {X 0,Y 608.449,Z 247.318,A -85,B 0,C 180,E1 -384.572,E2 -384.572} C_VEL
LIN {X 0,Y 608.428,Z 247.316,A -85,B 0,C 180,E1 -387.519,E2 -387.519} C_VEL
LIN {X 0,Y 608.444,Z 247.313,A -85,B 0,C 180,E1 -389.971,E2 -389.971} C_VEL
LIN {X 0,Y 608.447,Z 247.323,A -85,B 0,C 180,E1 -392.88,E2 -392.88} C_VEL
LIN {X 0,Y 608.426,Z 247.319,A -85,B 0,C 180,E1 -395.279,E2 -395.279} C_VEL
LIN {X 0,Y 608.45,Z 247.312,A -85,B 0,C 180,E1 -397.748,E2 -397.748} C_VEL
LIN {X 0,Y 608.448,Z 247.316,A -85,B 0,C 180,E1 -400.331,E2 -400.331} C_VEL
LIN {X 0,Y 608.439,Z 247.321,A -85,B 0,C 180,E1 -402.961,E2 -402.961} C_VEL
LIN {X 0,Y 608.432,Z 247.315,A -85,B 0,C 180,E1 -405.739,E2 -405.739} C_VEL
LIN {X 0,Y 608.446,Z 247.313,A -85,B 0,C 180,E1 -407.939,E2 -407.939} C_VEL
LIN {X 0,Y 608.469,Z 247.321,A -85,B 0,C 180,E1 -410.703,E2 -410.703} C_VEL
LIN {X 0,Y 608.432,Z 247.319,A -85,B 0,C 180,E1 -413.085,E2 -413.085} C_VEL
LIN {X 0,Y 608.443,Z 247.314,A -85,B 0,C 180,E1 -415.531,E2 -415.531} C_VEL
LIN {X 0,Y 608.448,Z 247.313,A -85,B 0,C 180,E1 -417.906,E2 -417.906} C_VEL
LIN {X 0,Y 608.482,Z 247.312,A -85,B 0,C 180,E1 -420.223,E2 -420.223} C_VEL
LIN {X 0,Y 608.422,Z 247.32,A -85,B 0,C 180,E1 -423.226,E2 -423.226} C_VEL
LIN {X 0,Y 608.437,Z 247.415,A -85,B 0,C 180,E1 -423.573,E2 -423.573} C_VEL
LIN {X 0,Y 608.731,Z 252.1,A -85,B 0,C 180,E1 -424.105,E2 -424.105} C_VEL
LIN {X 0,Y 608.661,Z 277.612,A -85,B 0,C 180,E1 -426.886,E2 -426.886} C_VEL
LIN {X 0,Y 608.602,Z 304.269,A -85,B 0,C 180,E1 -429.732,E2 -429.732} C_VEL
LIN {X 0,Y 608.575,Z 321.425,A -85,B 0,C 180,E1 -431.537,E2 -431.537} C_VEL
LIN {X 0,Y 608.762,Z 354.462,A -85,B 0,C 180,E1 -431.948,E2 -431.948} C_VEL
LIN {X 0,Y 608.682,Z 488.149,A -85,B 0,C 180,E1 -433.581,E2 -433.581} C_VEL
LIN {X 0,Y 608.65,Z 503.755,A -85,B 0,C 180,E1 -433.912,E2 -433.912} C_VEL
LIN {X 0,Y 608.618,Z 519.08,A -85,B 0,C 180,E1 -434.384,E2 -434.384} C_VEL
LIN {X 0,Y 608.606,Z 532.782,A -85,B 0,C 180,E1 -434.942,E2 -434.942} C_VEL
LIN {X 0,Y 608.575,Z 546.257,A -85,B 0,C 180,E1 -435.625,E2 -435.625} C_VEL
LIN {X 0,Y 608.554,Z 558.681,A -85,B 0,C 180,E1 -436.392,E2 -436.392} C_VEL
LIN {X 0,Y 608.528,Z 571.296,A -85,B 0,C 180,E1 -437.325,E2 -437.325} C_VEL
LIN {X 0,Y 608.496,Z 582.759,A -85,B 0,C 180,E1 -438.34,E2 -438.34} C_VEL
LIN {X 0,Y 608.476,Z 592.397,A -85,B 0,C 180,E1 -439.351,E2 -439.351} C_VEL
LIN {X 0,Y 608.477,Z 601.861,A -85,B 0,C 180,E1 -440.528,E2 -440.528} C_VEL
LIN {X 0,Y 608.455,Z 609.735,A -85,B 0,C 180,E1 -441.7,E2 -441.7} C_VEL
LIN {X 0,Y 608.441,Z 617.092,A -85,B 0,C 180,E1 -443.035,E2 -443.035} C_VEL
LIN {X 0,Y 608.449,Z 622.927,A -85,B 0,C 180,E1 -444.367,E2 -444.367} C_VEL
LIN {X 0,Y 608.427,Z 626.386,A -85,B 0,C 180,E1 -445.363,E2 -445.363} C_VEL
LIN {X 0,Y 608.421,Z 629.888,A -85,B 0,C 180,E1 -446.69,E2 -446.69} C_VEL
LIN {X 0,Y 608.442,Z 632.192,A -85,B 0,C 180,E1 -448.015,E2 -448.015} C_VEL
LIN {X 0,Y 608.436,Z 633.351,A -85,B 0,C 180,E1 -449.339,E2 -449.339} C_VEL
LIN {X 0,Y 608.436,Z 633.35,A -85,B 0,C 180,E1 -450.663,E2 -450.663} C_VEL
LIN {X 0,Y 608.442,Z 632.19,A -85,B 0,C 180,E1 -451.987,E2 -451.987} C_VEL
LIN {X 0,Y 608.421,Z 629.884,A -85,B 0,C 180,E1 -453.312,E2 -453.312} C_VEL
LIN {X 0,Y 608.427,Z 626.38,A -85,B 0,C 180,E1 -454.639,E2 -454.639} C_VEL
LIN {X 0,Y 608.431,Z 621.604,A -85,B 0,C 180,E1 -455.968,E2 -455.968} C_VEL
LIN {X 0,Y 608.458,Z 615.421,A -85,B 0,C 180,E1 -457.3,E2 -457.3} C_VEL
LIN {X 0,Y 608.465,Z 607.648,A -85,B 0,C 180,E1 -458.637,E2 -458.637} C_VEL
LIN {X 0,Y 608.471,Z 599.364,A -85,B 0,C 180,E1 -459.81,E2 -459.81} C_VEL
LIN {X 0,Y 608.493,Z 588.647,A -85,B 0,C 180,E1 -461.064,E2 -461.064} C_VEL
LIN {X 0,Y 608.522,Z 577.265,A -85,B 0,C 180,E1 -462.169,E2 -462.169} C_VEL
LIN {X 0,Y 608.548,Z 565.843,A -85,B 0,C 180,E1 -463.1,E2 -463.1} C_VEL
LIN {X 0,Y 608.565,Z 553.434,A -85,B 0,C 180,E1 -463.951,E2 -463.951} C_VEL
LIN {X 0,Y 608.569,Z 539.843,A -85,B 0,C 180,E1 -464.719,E2 -464.719} C_VEL
LIN {X 0,Y 608.634,Z 525.771,A -85,B 0,C 180,E1 -465.36,E2 -465.36} C_VEL
LIN {X 0,Y 608.637,Z 511.276,A -85,B 0,C 180,E1 -465.875,E2 -465.875} C_VEL
LIN {X 0,Y 608.689,Z 495.979,A -85,B 0,C 180,E1 -466.27,E2 -466.27} C_VEL
LIN {X 0,Y 608.689,Z 480.006,A -85,B 0,C 180,E1 -466.535,E2 -466.535} C_VEL
LIN {X 0,Y 608.63,Z 321.907,A -85,B 0,C 180,E1 -468.453,E2 -468.453} C_VEL
LIN {X 0,Y 608.571,Z 321.123,A -85,B 0,C 180,E1 -468.495,E2 -468.495} C_VEL
LIN {X 0,Y 608.621,Z 295.921,A -85,B 0,C 180,E1 -471.154,E2 -471.154} C_VEL
LIN {X 0,Y 608.698,Z 268.823,A -85,B 0,C 180,E1 -474.065,E2 -474.065} C_VEL
LIN {X 0,Y 608.721,Z 249.271,A -85,B 0,C 180,E1 -476.208,E2 -476.208} C_VEL
LIN {X 0,Y 608.434,Z 247.318,A -85,B 0,C 180,E1 -476.452,E2 -476.452} C_VEL
LIN {X 0,Y 608.431,Z 247.322,A -85,B 0,C 180,E1 -479.023,E2 -479.023} C_VEL
LIN {X 0,Y 608.464,Z 247.32,A -85,B 0,C 180,E1 -481.317,E2 -481.317} C_VEL
LIN {X 0,Y 608.477,Z 247.312,A -85,B 0,C 180,E1 -483.735,E2 -483.735} C_VEL
LIN {X 0,Y 608.446,Z 247.314,A -85,B 0,C 180,E1 -486.093,E2 -486.093} C_VEL
LIN {X 0,Y 608.442,Z 247.318,A -85,B 0,C 180,E1 -488.591,E2 -488.591} C_VEL
LIN {X 0,Y 608.462,Z 247.315,A -85,B 0,C 180,E1 -491.342,E2 -491.342} C_VEL
LIN {X 0,Y 608.448,Z 247.315,A -85,B 0,C 180,E1 -494.263,E2 -494.263} C_VEL
LIN {X 0,Y 608.454,Z 247.318,A -85,B 0,C 180,E1 -497.04,E2 -497.04} C_VEL
LIN {X 0,Y 608.458,Z 247.312,A -85,B 0,C 180,E1 -499.697,E2 -499.697} C_VEL
LIN {X 0,Y 608.468,Z 247.315,A -85,B 0,C 180,E1 -502.253,E2 -502.253} C_VEL
LIN {X 0,Y 608.438,Z 247.317,A -85,B 0,C 180,E1 -505.097,E2 -505.097} C_VEL
LIN {X 0,Y 608.462,Z 247.311,A -85,B 0,C 180,E1 -507.478,E2 -507.478} C_VEL
LIN {X 0,Y 608.474,Z 247.317,A -85,B 0,C 180,E1 -510.221,E2 -510.221} C_VEL
LIN {X 0,Y 608.461,Z 247.315,A -85,B 0,C 180,E1 -512.797,E2 -512.797} C_VEL
LIN {X 0,Y 608.447,Z 247.314,A -85,B 0,C 180,E1 -515.428,E2 -515.428} C_VEL
LIN {X 0,Y 608.458,Z 247.321,A -85,B 0,C 180,E1 -518.308,E2 -518.308} C_VEL
LIN {X 0,Y 608.452,Z 247.357,A -85,B 0,C 180,E1 -519.326,E2 -519.326} C_VEL
LIN {X 0,Y 608.535,Z 263.5,A -85,B 0,C 180,E1 -521.607,E2 -521.607} C_VEL
LIN {X 0,Y 608.76,Z 270.014,A -85,B 0,C 180,E1 -521.695,E2 -521.695} C_VEL
LIN {X 0,Y 608.694,Z 428.356,A -85,B 0,C 180,E1 -523.63,E2 -523.63} C_VEL
LIN {X 0,Y 608.667,Z 444.396,A -85,B 0,C 180,E1 -523.976,E2 -523.976} C_VEL
LIN {X 0,Y 608.652,Z 458.979,A -85,B 0,C 180,E1 -524.427,E2 -524.427} C_VEL
LIN {X 0,Y 608.589,Z 473.656,A -85,B 0,C 180,E1 -525.025,E2 -525.025} C_VEL
LIN {X 0,Y 608.577,Z 487.425,A -85,B 0,C 180,E1 -525.734,E2 -525.734} C_VEL
LIN {X 0,Y 608.548,Z 500.541,A -85,B 0,C 180,E1 -526.56,E2 -526.56} C_VEL
LIN {X 0,Y 608.505,Z 512.83,A -85,B 0,C 180,E1 -527.493,E2 -527.493} C_VEL
LIN {X 0,Y 608.498,Z 524.048,A -85,B 0,C 180,E1 -528.507,E2 -528.507} C_VEL
LIN {X 0,Y 608.478,Z 534.933,A -85,B 0,C 180,E1 -529.686,E2 -529.686} C_VEL
LIN {X 0,Y 608.469,Z 543.979,A -85,B 0,C 180,E1 -530.861,E2 -530.861} C_VEL
LIN {X 0,Y 608.454,Z 551.477,A -85,B 0,C 180,E1 -532.032,E2 -532.032} C_VEL
LIN {X 0,Y 608.447,Z 558.628,A -85,B 0,C 180,E1 -533.396,E2 -533.396} C_VEL
LIN {X 0,Y 608.435,Z 563.991,A -85,B 0,C 180,E1 -534.697,E2 -534.697} C_VEL
LIN {X 0,Y 608.427,Z 568.167,A -85,B 0,C 180,E1 -536.025,E2 -536.025} C_VEL
LIN {X 0,Y 608.42,Z 571.108,A -85,B 0,C 180,E1 -537.351,E2 -537.351} C_VEL
LIN {X 0,Y 608.448,Z 572.881,A -85,B 0,C 180,E1 -538.676,E2 -538.676} C_VEL
LIN {X 0,Y 608.431,Z 573.495,A -85,B 0,C 180,E1 -539.999,E2 -539.999} C_VEL
LIN {X 0,Y 608.445,Z 572.945,A -85,B 0,C 180,E1 -541.323,E2 -541.323} C_VEL
LIN {X 0,Y 608.424,Z 571.26,A -85,B 0,C 180,E1 -542.648,E2 -542.648} C_VEL
LIN {X 0,Y 608.429,Z 568.41,A -85,B 0,C 180,E1 -543.974,E2 -543.974} C_VEL
LIN {X 0,Y 608.435,Z 564.33,A -85,B 0,C 180,E1 -545.302,E2 -545.302} C_VEL
LIN {X 0,Y 608.44,Z 558.926,A -85,B 0,C 180,E1 -546.632,E2 -546.632} C_VEL
LIN {X 0,Y 608.456,Z 552.024,A -85,B 0,C 180,E1 -547.967,E2 -547.967} C_VEL
LIN {X 0,Y 608.464,Z 544.491,A -85,B 0,C 180,E1 -549.153,E2 -549.153} C_VEL
LIN {X 0,Y 607.763,Z 541.257,A -85,B 0,C 180,E1 -549.614,E2 -549.614} C_VEL
LIN {X 0,Y 604.898,Z 535.859,A -85,B 0,C 180,E1 -550.354,E2 -550.354} C_VEL
LIN {X 0,Y 602.083,Z 530.099,A -85,B 0,C 180,E1 -551.071,E2 -551.071} C_VEL
LIN {X 0,Y 601.459,Z 526.221,A -85,B 0,C 180,E1 -551.494,E2 -551.494} C_VEL
LIN {X 0,Y 601.492,Z 515.856,A -85,B 0,C 180,E1 -552.483,E2 -552.483} C_VEL
LIN {X 0,Y 601.577,Z 504.152,A -85,B 0,C 180,E1 -553.425,E2 -553.425} C_VEL
LIN {X 0,Y 601.627,Z 491.376,A -85,B 0,C 180,E1 -554.286,E2 -554.286} C_VEL
LIN {X 0,Y 601.685,Z 477.292,A -85,B 0,C 180,E1 -555.063,E2 -555.063} C_VEL
LIN {X 0,Y 601.755,Z 462.499,A -85,B 0,C 180,E1 -555.712,E2 -555.712} C_VEL
LIN {X 0,Y 601.81,Z 446.846,A -85,B 0,C 180,E1 -556.232,E2 -556.232} C_VEL
LIN {X 0,Y 601.877,Z 431.595,A -85,B 0,C 180,E1 -556.59,E2 -556.59} C_VEL
LIN {X 0,Y 601.88,Z 411.427,A -85,B 0,C 180,E1 -556.877,E2 -556.877} C_VEL
LIN {X 0,Y 601.937,Z 265.484,A -85,B 0,C 180,E1 -558.666,E2 -558.666} C_VEL
LIN {X 0,Y 601.531,Z 263.403,A -85,B 0,C 180,E1 -558.719,E2 -558.719} C_VEL
LIN {X 0,Y 601.491,Z 248.764,A -85,B 0,C 180,E1 -560.812,E2 -560.812} C_VEL
LIN {X 0,Y 601.41,Z 248.193,A -85,B 0,C 180,E1 -560.901,E2 -560.901} C_VEL
LIN {X 0,Y 601.394,Z 248.195,A -85,B 0,C 180,E1 -563.411,E2 -563.411} C_VEL
LIN {X 0,Y 601.39,Z 248.196,A -85,B 0,C 180,E1 -566.364,E2 -566.364} C_VEL
LIN {X 0,Y 601.411,Z 248.19,A -85,B 0,C 180,E1 -568.784,E2 -568.784} C_VEL
LIN {X 0,Y 601.418,Z 248.192,A -85,B 0,C 180,E1 -571.454,E2 -571.454} C_VEL
LIN {X 0,Y 601.421,Z 248.195,A -85,B 0,C 180,E1 -574.118,E2 -574.118} C_VEL
LIN {X 0,Y 601.391,Z 248.193,A -85,B 0,C 180,E1 -576.583,E2 -576.583} C_VEL
LIN {X 0,Y 601.415,Z 248.194,A -85,B 0,C 180,E1 -579.532,E2 -579.532} C_VEL
LIN {X 0,Y 601.419,Z 248.198,A -85,B 0,C 180,E1 -581.764,E2 -581.764} C_VEL
LIN {X 0,Y 601.448,Z 248.191,A -85,B 0,C 180,E1 -583.583,E2 -583.583} C_VEL
LIN {X 0,Y 601.403,Z 248.192,A -85,B 0,C 180,E1 -586.429,E2 -586.429} C_VEL
LIN {X 0,Y 601.404,Z 248.191,A -85,B 0,C 180,E1 -589.124,E2 -589.124} C_VEL
LIN {X 0,Y 601.419,Z 248.198,A -85,B 0,C 180,E1 -591.731,E2 -591.731} C_VEL
LIN {X 0,Y 601.379,Z 248.196,A -85,B 0,C 180,E1 -594.244,E2 -594.244} C_VEL
LIN {X 0,Y 601.409,Z 248.19,A -85,B 0,C 180,E1 -596.685,E2 -596.685} C_VEL
LIN {X 0,Y 601.41,Z 248.191,A -85,B 0,C 180,E1 -599.057,E2 -599.057} C_VEL
LIN {X 0,Y 601.437,Z 248.191,A -85,B 0,C 180,E1 -601.373,E2 -601.373} C_VEL
LIN {X 0,Y 601.39,Z 248.196,A -85,B 0,C 180,E1 -604.135,E2 -604.135} C_VEL
LIN {X 0,Y 601.385,Z 248.193,A -85,B 0,C 180,E1 -606.588,E2 -606.588} C_VEL
LIN {X 0,Y 601.431,Z 248.194,A -85,B 0,C 180,E1 -609.477,E2 -609.477} C_VEL
LIN {X 0,Y 601.379,Z 248.195,A -85,B 0,C 180,E1 -612.31,E2 -612.31} C_VEL
LIN {X 0,Y 601.397,Z 248.192,A -85,B 0,C 180,E1 -614.408,E2 -614.408} C_VEL
LIN {X 0,Y 601.415,Z 248.192,A -85,B 0,C 180,E1 -617.171,E2 -617.171} C_VEL
LIN {X 0,Y 601.416,Z 248.194,A -85,B 0,C 180,E1 -619.904,E2 -619.904} C_VEL
LIN {X 0,Y 601.428,Z 248.187,A -85,B 0,C 180,E1 -622.614,E2 -622.614} C_VEL
LIN {X 0,Y 601.424,Z 248.194,A -85,B 0,C 180,E1 -625.307,E2 -625.307} C_VEL
LIN {X 0,Y 601.402,Z 248.194,A -85,B 0,C 180,E1 -627.99,E2 -627.99} C_VEL
LIN {X 0,Y 601.421,Z 248.192,A -85,B 0,C 180,E1 -629.999,E2 -629.999} C_VEL
LIN {X 0,Y 601.425,Z 248.188,A -85,B 0,C 180,E1 -632.678,E2 -632.678} C_VEL
LIN {X 0,Y 601.429,Z 248.195,A -85,B 0,C 180,E1 -635.363,E2 -635.363} C_VEL
LIN {X 0,Y 601.421,Z 248.19,A -85,B 0,C 180,E1 -638.06,E2 -638.06} C_VEL
LIN {X 0,Y 601.416,Z 248.192,A -85,B 0,C 180,E1 -641.013,E2 -641.013} C_VEL
LIN {X 0,Y 601.409,Z 248.2,A -85,B 0,C 180,E1 -643.515,E2 -643.515} C_VEL
LIN {X 0,Y 601.415,Z 248.189,A -85,B 0,C 180,E1 -646.286,E2 -646.286} C_VEL
LIN {X 0,Y 601.408,Z 248.195,A -85,B 0,C 180,E1 -649.098,E2 -649.098} C_VEL
LIN {X 0,Y 601.403,Z 248.198,A -85,B 0,C 180,E1 -651.238,E2 -651.238} C_VEL
LIN {X 0,Y 601.427,Z 248.188,A -85,B 0,C 180,E1 -654.14,E2 -654.14} C_VEL
LIN {X 0,Y 601.451,Z 248.19,A -85,B 0,C 180,E1 -657.11,E2 -657.11} C_VEL
LIN {X 0,Y 601.405,Z 248.201,A -85,B 0,C 180,E1 -659.392,E2 -659.392} C_VEL
LIN {X 0,Y 601.396,Z 248.196,A -85,B 0,C 180,E1 -661.726,E2 -661.726} C_VEL
LIN {X 0,Y 601.416,Z 248.189,A -85,B 0,C 180,E1 -664.118,E2 -664.118} C_VEL
LIN {X 0,Y 601.396,Z 248.192,A -85,B 0,C 180,E1 -666.582,E2 -666.582} C_VEL
LIN {X 0,Y 601.425,Z 248.194,A -85,B 0,C 180,E1 -669.535,E2 -669.535} C_VEL
LIN {X 0,Y 601.404,Z 248.193,A -85,B 0,C 180,E1 -671.765,E2 -671.765} C_VEL
LIN {X 0,Y 601.409,Z 248.19,A -85,B 0,C 180,E1 -674.535,E2 -674.535} C_VEL
LIN {X 0,Y 601.4,Z 248.201,A -85,B 0,C 180,E1 -677.33,E2 -677.33} C_VEL
LIN {X 0,Y 601.395,Z 248.192,A -85,B 0,C 180,E1 -680.005,E2 -680.005} C_VEL
LIN {X 0,Y 601.424,Z 248.189,A -85,B 0,C 180,E1 -682.617,E2 -682.617} C_VEL
LIN {X 0,Y 601.438,Z 248.194,A -85,B 0,C 180,E1 -685.071,E2 -685.071} C_VEL
LIN {X 0,Y 601.412,Z 248.195,A -85,B 0,C 180,E1 -687.484,E2 -687.484} C_VEL
LIN {X 0,Y 601.411,Z 248.191,A -85,B 0,C 180,E1 -689.852,E2 -689.852} C_VEL
LIN {X 0,Y 601.41,Z 248.192,A -85,B 0,C 180,E1 -692.636,E2 -692.636} C_VEL
LIN {X 0,Y 601.392,Z 248.202,A -85,B 0,C 180,E1 -695.122,E2 -695.122} C_VEL
LIN {X 0,Y 601.4,Z 248.197,A -85,B 0,C 180,E1 -697.394,E2 -697.394} C_VEL
LIN {X 0,Y 601.39,Z 248.192,A -85,B 0,C 180,E1 -700.191,E2 -700.191} C_VEL
LIN {X 0,Y 601.421,Z 248.197,A -85,B 0,C 180,E1 -703.015,E2 -703.015} C_VEL
LIN {X 0,Y 601.385,Z 248.193,A -85,B 0,C 180,E1 -705.916,E2 -705.916} C_VEL
LIN {X 0,Y 601.425,Z 248.19,A -85,B 0,C 180,E1 -708.542,E2 -708.542} C_VEL
LIN {X 0,Y 601.4,Z 248.198,A -85,B 0,C 180,E1 -711.262,E2 -711.262} C_VEL
LIN {X 0,Y 601.416,Z 248.194,A -85,B 0,C 180,E1 -713.345,E2 -713.345} C_VEL
LIN {X 0,Y 601.376,Z 248.194,A -85,B 0,C 180,E1 -715.98,E2 -715.98} C_VEL
LIN {X 0,Y 601.428,Z 248.192,A -85,B 0,C 180,E1 -718.661,E2 -718.661} C_VEL
LIN {X 0,Y 601.405,Z 248.195,A -85,B 0,C 180,E1 -721.34,E2 -721.34} C_VEL
LIN {X 0,Y 601.413,Z 248.194,A -85,B 0,C 180,E1 -723.35,E2 -723.35} C_VEL
LIN {X 0,Y 601.384,Z 248.193,A -85,B 0,C 180,E1 -726.038,E2 -726.038} C_VEL
LIN {X 0,Y 601.432,Z 248.193,A -85,B 0,C 180,E1 -728.738,E2 -728.738} C_VEL
LIN {X 0,Y 601.418,Z 248.191,A -85,B 0,C 180,E1 -731.459,E2 -731.459} C_VEL
LIN {X 0,Y 601.408,Z 248.19,A -85,B 0,C 180,E1 -734.206,E2 -734.206} C_VEL
LIN {X 0,Y 601.421,Z 248.198,A -85,B 0,C 180,E1 -736.987,E2 -736.987} C_VEL
LIN {X 0,Y 601.387,Z 248.192,A -85,B 0,C 180,E1 -739.81,E2 -739.81} C_VEL
LIN {X 0,Y 601.448,Z 248.191,A -85,B 0,C 180,E1 -742.617,E2 -742.617} C_VEL
LIN {X 0,Y 601.39,Z 248.203,A -85,B 0,C 180,E1 -744.879,E2 -744.879} C_VEL
LIN {X 0,Y 601.388,Z 248.195,A -85,B 0,C 180,E1 -747.36,E2 -747.36} C_VEL
LIN {X 0,Y 601.399,Z 248.193,A -85,B 0,C 180,E1 -749.394,E2 -749.394} C_VEL
LIN {X 0,Y 601.392,Z 248.192,A -85,B 0,C 180,E1 -751.728,E2 -751.728} C_VEL
LIN {X 0,Y 601.414,Z 248.19,A -85,B 0,C 180,E1 -754.12,E2 -754.12} C_VEL
LIN {X 0,Y 601.423,Z 248.19,A -85,B 0,C 180,E1 -757.383,E2 -757.383} C_VEL
LIN {X 0,Y 601.392,Z 248.192,A -85,B 0,C 180,E1 -759.997,E2 -759.997} C_VEL
LIN {X 0,Y 601.406,Z 248.199,A -85,B 0,C 180,E1 -762.671,E2 -762.671} C_VEL
LIN {X 0,Y 601.39,Z 248.193,A -85,B 0,C 180,E1 -765.48,E2 -765.48} C_VEL
LIN {X 0,Y 601.375,Z 248.195,A -85,B 0,C 180,E1 -767.413,E2 -767.413} C_VEL
LIN {X 0,Y 601.405,Z 248.191,A -85,B 0,C 180,E1 -770.006,E2 -770.006} C_VEL
LIN {X 0,Y 601.429,Z 248.197,A -85,B 0,C 180,E1 -772.619,E2 -772.619} C_VEL
LIN {X 0,Y 601.389,Z 248.196,A -85,B 0,C 180,E1 -775.068,E2 -775.068} C_VEL
LIN {X 0,Y 601.4,Z 248.191,A -85,B 0,C 180,E1 -777.484,E2 -777.484} C_VEL
LIN {X 0,Y 601.399,Z 248.192,A -85,B 0,C 180,E1 -779.857,E2 -779.857} C_VEL
LIN {X 0,Y 601.438,Z 248.195,A -85,B 0,C 180,E1 -782.89,E2 -782.89} C_VEL
LIN {X 0,Y 601.404,Z 248.248,A -85,B 0,C 180,E1 -783.334,E2 -783.334} C_VEL
LIN {X 0,Y 601.976,Z 252.565,A -85,B 0,C 180,E1 -783.845,E2 -783.845} C_VEL
LIN {X 0,Y 601.856,Z 277.612,A -85,B 0,C 180,E1 -786.609,E2 -786.609} C_VEL
LIN {X 0,Y 601.744,Z 304.269,A -85,B 0,C 180,E1 -789.491,E2 -789.491} C_VEL
LIN {X 0,Y 601.654,Z 321.453,A -85,B 0,C 180,E1 -791.319,E2 -791.319} C_VEL
LIN {X 0,Y 602.036,Z 325.99,A -85,B 0,C 180,E1 -791.388,E2 -791.388} C_VEL
LIN {X 0,Y 601.878,Z 488.509,A -85,B 0,C 180,E1 -793.397,E2 -793.397} C_VEL
LIN {X 0,Y 601.829,Z 503.753,A -85,B 0,C 180,E1 -793.725,E2 -793.725} C_VEL
LIN {X 0,Y 601.767,Z 519.078,A -85,B 0,C 180,E1 -794.202,E2 -794.202} C_VEL
LIN {X 0,Y 601.719,Z 532.785,A -85,B 0,C 180,E1 -794.765,E2 -794.765} C_VEL
LIN {X 0,Y 601.661,Z 546.253,A -85,B 0,C 180,E1 -795.456,E2 -795.456} C_VEL
LIN {X 0,Y 601.617,Z 559.46,A -85,B 0,C 180,E1 -796.284,E2 -796.284} C_VEL
LIN {X 0,Y 601.532,Z 571.298,A -85,B 0,C 180,E1 -797.175,E2 -797.175} C_VEL
LIN {X 0,Y 601.487,Z 582.759,A -85,B 0,C 180,E1 -798.202,E2 -798.202} C_VEL
LIN {X 0,Y 601.431,Z 592.398,A -85,B 0,C 180,E1 -799.225,E2 -799.225} C_VEL
LIN {X 0,Y 601.428,Z 601.862,A -85,B 0,C 180,E1 -800.416,E2 -800.416} C_VEL
LIN {X 0,Y 601.368,Z 609.736,A -85,B 0,C 180,E1 -801.601,E2 -801.601} C_VEL
LIN {X 0,Y 601.368,Z 617.092,A -85,B 0,C 180,E1 -802.952,E2 -802.952} C_VEL
LIN {X 0,Y 601.371,Z 622.927,A -85,B 0,C 180,E1 -804.3,E2 -804.3} C_VEL
LIN {X 0,Y 601.33,Z 626.386,A -85,B 0,C 180,E1 -805.308,E2 -805.308} C_VEL
LIN {X 0,Y 601.337,Z 629.888,A -85,B 0,C 180,E1 -806.651,E2 -806.651} C_VEL
LIN {X 0,Y 601.341,Z 632.193,A -85,B 0,C 180,E1 -807.992,E2 -807.992} C_VEL
LIN {X 0,Y 601.337,Z 633.35,A -85,B 0,C 180,E1 -809.331,E2 -809.331} C_VEL
LIN {X 0,Y 601.337,Z 633.35,A -85,B 0,C 180,E1 -810.671,E2 -810.671} C_VEL
LIN {X 0,Y 601.341,Z 632.191,A -85,B 0,C 180,E1 -812.01,E2 -812.01} C_VEL
LIN {X 0,Y 601.337,Z 629.884,A -85,B 0,C 180,E1 -813.351,E2 -813.351} C_VEL
LIN {X 0,Y 601.33,Z 626.38,A -85,B 0,C 180,E1 -814.694,E2 -814.694} C_VEL
LIN {X 0,Y 601.352,Z 621.604,A -85,B 0,C 180,E1 -816.039,E2 -816.039} C_VEL
LIN {X 0,Y 601.366,Z 615.421,A -85,B 0,C 180,E1 -817.387,E2 -817.387} C_VEL
LIN {X 0,Y 601.388,Z 607.648,A -85,B 0,C 180,E1 -818.739,E2 -818.739} C_VEL
LIN {X 0,Y 601.427,Z 599.364,A -85,B 0,C 180,E1 -819.926,E2 -819.926} C_VEL
LIN {X 0,Y 601.461,Z 588.927,A -85,B 0,C 180,E1 -821.165,E2 -821.165} C_VEL
LIN {X 0,Y 601.514,Z 579.183,A -85,B 0,C 180,E1 -822.141,E2 -822.141} C_VEL
LIN {X 0,Y 601.571,Z 567.005,A -85,B 0,C 180,E1 -823.169,E2 -823.169} C_VEL
LIN {X 0,Y 601.609,Z 555.065,A -85,B 0,C 180,E1 -824.012,E2 -824.012} C_VEL
LIN {X 0,Y 601.67,Z 541.512,A -85,B 0,C 180,E1 -824.805,E2 -824.805} C_VEL
LIN {X 0,Y 601.766,Z 526.824,A -85,B 0,C 180,E1 -825.496,E2 -825.496} C_VEL
LIN {X 0,Y 601.788,Z 512.594,A -85,B 0,C 180,E1 -826.017,E2 -826.017} C_VEL
LIN {X 0,Y 601.86,Z 497.653,A -85,B 0,C 180,E1 -826.421,E2 -826.421} C_VEL
LIN {X 0,Y 601.871,Z 482.649,A -85,B 0,C 180,E1 -826.69,E2 -826.69} C_VEL
LIN {X 0,Y 601.928,Z 322.914,A -85,B 0,C 180,E1 -828.653,E2 -828.653} C_VEL
LIN {X 0,Y 601.666,Z 321.314,A -85,B 0,C 180,E1 -828.695,E2 -828.695} C_VEL
LIN {X 0,Y 601.749,Z 295.921,A -85,B 0,C 180,E1 -831.407,E2 -831.407} C_VEL
LIN {X 0,Y 601.888,Z 269.746,A -85,B 0,C 180,E1 -834.253,E2 -834.253} C_VEL
LIN {X 0,Y 601.942,Z 250.937,A -85,B 0,C 180,E1 -836.339,E2 -836.339} C_VEL
LIN {X 0,Y 601.387,Z 248.199,A -85,B 0,C 180,E1 -836.693,E2 -836.693} C_VEL
LIN {X 0,Y 601.409,Z 248.199,A -85,B 0,C 180,E1 -839.394,E2 -839.394} C_VEL
LIN {X 0,Y 601.404,Z 248.194,A -85,B 0,C 180,E1 -841.727,E2 -841.727} C_VEL
LIN {X 0,Y 601.426,Z 248.189,A -85,B 0,C 180,E1 -844.119,E2 -844.119} C_VEL
LIN {X 0,Y 601.405,Z 248.194,A -85,B 0,C 180,E1 -846.583,E2 -846.583} C_VEL
LIN {X 0,Y 601.446,Z 248.188,A -85,B 0,C 180,E1 -849.536,E2 -849.536} C_VEL
LIN {X 0,Y 601.41,Z 248.196,A -85,B 0,C 180,E1 -852.59,E2 -852.59} C_VEL
LIN {X 0,Y 601.432,Z 248.189,A -85,B 0,C 180,E1 -855.482,E2 -855.482} C_VEL
LIN {X 0,Y 601.426,Z 248.193,A -85,B 0,C 180,E1 -858.407,E2 -858.407} C_VEL
LIN {X 0,Y 601.406,Z 248.197,A -85,B 0,C 180,E1 -860.873,E2 -860.873} C_VEL
LIN {X 0,Y 601.397,Z 248.192,A -85,B 0,C 180,E1 -863.416,E2 -863.416} C_VEL
LIN {X 0,Y 601.437,Z 248.19,A -85,B 0,C 180,E1 -866.064,E2 -866.064} C_VEL
LIN {X 0,Y 601.422,Z 248.197,A -85,B 0,C 180,E1 -868.546,E2 -868.546} C_VEL
LIN {X 0,Y 601.426,Z 248.188,A -85,B 0,C 180,E1 -871.373,E2 -871.373} C_VEL
LIN {X 0,Y 601.42,Z 248.197,A -85,B 0,C 180,E1 -874.132,E2 -874.132} C_VEL
LIN {X 0,Y 601.391,Z 248.198,A -85,B 0,C 180,E1 -876.588,E2 -876.588} C_VEL
LIN {X 0,Y 601.425,Z 248.271,A -85,B 0,C 180,E1 -879.204,E2 -879.204} C_VEL
LIN {X 0,Y 601.545,Z 258.88,A -85,B 0,C 180,E1 -880.728,E2 -880.728} C_VEL
LIN {X 0,Y 601.575,Z 263.559,A -85,B 0,C 180,E1 -881.388,E2 -881.388} C_VEL
LIN {X 0,Y 602.043,Z 266.617,A -85,B 0,C 180,E1 -881.441,E2 -881.441} C_VEL
LIN {X 0,Y 601.89,Z 427.777,A -85,B 0,C 180,E1 -883.431,E2 -883.431} C_VEL
LIN {X 0,Y 601.833,Z 443.608,A -85,B 0,C 180,E1 -883.767,E2 -883.767} C_VEL
LIN {X 0,Y 601.782,Z 457.715,A -85,B 0,C 180,E1 -884.201,E2 -884.201} C_VEL
LIN {X 0,Y 601.73,Z 471.742,A -85,B 0,C 180,E1 -884.764,E2 -884.764} C_VEL
LIN {X 0,Y 601.666,Z 485.395,A -85,B 0,C 180,E1 -885.455,E2 -885.455} C_VEL
LIN {X 0,Y 601.617,Z 498.796,A -85,B 0,C 180,E1 -886.284,E2 -886.284} C_VEL
LIN {X 0,Y 601.532,Z 510.715,A -85,B 0,C 180,E1 -887.174,E2 -887.174} C_VEL
LIN {X 0,Y 601.489,Z 522.284,A -85,B 0,C 180,E1 -888.201,E2 -888.201} C_VEL
LIN {X 0,Y 601.43,Z 531.991,A -85,B 0,C 180,E1 -889.224,E2 -889.224} C_VEL
LIN {X 0,Y 601.43,Z 541.527,A -85,B 0,C 180,E1 -890.414,E2 -890.414} C_VEL
LIN {X 0,Y 601.4,Z 550.469,A -85,B 0,C 180,E1 -891.769,E2 -891.769} C_VEL
LIN {X 0,Y 601.37,Z 556.874,A -85,B 0,C 180,E1 -892.951,E2 -892.951} C_VEL
LIN {X 0,Y 601.369,Z 562.756,A -85,B 0,C 180,E1 -894.299,E2 -894.299} C_VEL
LIN {X 0,Y 601.328,Z 566.243,A -85,B 0,C 180,E1 -895.307,E2 -895.307} C_VEL
LIN {X 0,Y 601.34,Z 569.789,A -85,B 0,C 180,E1 -896.649,E2 -896.649} C_VEL
LIN {X 0,Y 601.337,Z 572.141,A -85,B 0,C 180,E1 -897.99,E2 -897.99} C_VEL
LIN {X 0,Y 601.335,Z 573.332,A -85,B 0,C 180,E1 -899.33,E2 -899.33} C_VEL
LIN {X 0,Y 601.338,Z 573.361,A -85,B 0,C 180,E1 -900.669,E2 -900.669} C_VEL
LIN {X 0,Y 601.341,Z 572.247,A -85,B 0,C 180,E1 -902.009,E2 -902.009} C_VEL
LIN {X 0,Y 601.341,Z 569.984,A -85,B 0,C 180,E1 -903.349,E2 -903.349} C_VEL
LIN {X 0,Y 601.332,Z 566.53,A -85,B 0,C 180,E1 -904.692,E2 -904.692} C_VEL
LIN {X 0,Y 601.353,Z 561.8,A -85,B 0,C 180,E1 -906.037,E2 -906.037} C_VEL
LIN {X 0,Y 601.365,Z 555.663,A -85,B 0,C 180,E1 -907.385,E2 -907.385} C_VEL
LIN {X 0,Y 601.39,Z 547.955,A -85,B 0,C 180,E1 -908.738,E2 -908.738} C_VEL
LIN {X 0,Y 601.427,Z 539.706,A -85,B 0,C 180,E1 -909.925,E2 -909.925} C_VEL
LIN {X 0,Y 601.443,Z 529.374,A -85,B 0,C 180,E1 -911.164,E2 -911.164} C_VEL
LIN {X 0,Y 601.459,Z 526.221,A -85,B 0,C 180,E1 -911.494,E2 -911.494} C_VEL
LIN {X 0,Y 600.839,Z 522.262,A -85,B 0,C 180,E1 -911.908,E2 -911.908} C_VEL
LIN {X 0,Y 598.052,Z 515.75,A -85,B 0,C 180,E1 -912.572,E2 -912.572} C_VEL
LIN {X 0,Y 595.246,Z 508.903,A -85,B 0,C 180,E1 -913.206,E2 -913.206} C_VEL
LIN {X 0,Y 594.595,Z 504.378,A -85,B 0,C 180,E1 -913.569,E2 -913.569} C_VEL
LIN {X 0,Y 594.7,Z 491.371,A -85,B 0,C 180,E1 -914.456,E2 -914.456} C_VEL
LIN {X 0,Y 594.801,Z 477.286,A -85,B 0,C 180,E1 -915.241,E2 -915.241} C_VEL
LIN {X 0,Y 594.905,Z 462.493,A -85,B 0,C 180,E1 -915.897,E2 -915.897} C_VEL
LIN {X 0,Y 594.973,Z 446.829,A -85,B 0,C 180,E1 -916.424,E2 -916.424} C_VEL
LIN {X 0,Y 595.08,Z 432.15,A -85,B 0,C 180,E1 -916.774,E2 -916.774} C_VEL
LIN {X 0,Y 595.099,Z 412.975,A -85,B 0,C 180,E1 -917.056,E2 -917.056} C_VEL
LIN {X 0,Y 595.224,Z 266.682,A -85,B 0,C 180,E1 -918.869,E2 -918.869} C_VEL
LIN {X 0,Y 594.581,Z 263.498,A -85,B 0,C 180,E1 -918.932,E2 -918.932} C_VEL
LIN {X 0,Y 594.629,Z 250.802,A -85,B 0,C 180,E1 -920.767,E2 -920.767} C_VEL
LIN {X 0,Y 594.378,Z 249.071,A -85,B 0,C 180,E1 -921.042,E2 -921.042} C_VEL
LIN {X 0,Y 594.365,Z 249.075,A -85,B 0,C 180,E1 -923.704,E2 -923.704} C_VEL
LIN {X 0,Y 594.363,Z 249.077,A -85,B 0,C 180,E1 -926.017,E2 -926.017} C_VEL
LIN {X 0,Y 594.361,Z 249.073,A -85,B 0,C 180,E1 -928.227,E2 -928.227} C_VEL
LIN {X 0,Y 594.366,Z 249.068,A -85,B 0,C 180,E1 -930.56,E2 -930.56} C_VEL
LIN {X 0,Y 594.374,Z 249.066,A -85,B 0,C 180,E1 -932.949,E2 -932.949} C_VEL
LIN {X 0,Y 594.346,Z 249.072,A -85,B 0,C 180,E1 -935.408,E2 -935.408} C_VEL
LIN {X 0,Y 594.378,Z 249.075,A -85,B 0,C 180,E1 -937.94,E2 -937.94} C_VEL
LIN {X 0,Y 594.368,Z 249.067,A -85,B 0,C 180,E1 -940.82,E2 -940.82} C_VEL
LIN {X 0,Y 594.373,Z 249.077,A -85,B 0,C 180,E1 -943.839,E2 -943.839} C_VEL
LIN {X 0,Y 594.349,Z 249.069,A -85,B 0,C 180,E1 -946.698,E2 -946.698} C_VEL
LIN {X 0,Y 594.367,Z 249.071,A -85,B 0,C 180,E1 -949.432,E2 -949.432} C_VEL
LIN {X 0,Y 594.384,Z 249.066,A -85,B 0,C 180,E1 -952.391,E2 -952.391} C_VEL
LIN {X 0,Y 594.391,Z 249.069,A -85,B 0,C 180,E1 -955.42,E2 -955.42} C_VEL
LIN {X 0,Y 594.37,Z 249.068,A -85,B 0,C 180,E1 -958.357,E2 -958.357} C_VEL
LIN {X 0,Y 594.379,Z 249.066,A -85,B 0,C 180,E1 -961.041,E2 -961.041} C_VEL
LIN {X 0,Y 594.368,Z 249.073,A -85,B 0,C 180,E1 -963.979,E2 -963.979} C_VEL
LIN {X 0,Y 594.367,Z 249.069,A -85,B 0,C 180,E1 -966.294,E2 -966.294} C_VEL
LIN {X 0,Y 594.405,Z 249.065,A -85,B 0,C 180,E1 -969.224,E2 -969.224} C_VEL
LIN {X 0,Y 594.34,Z 249.074,A -85,B 0,C 180,E1 -972.094,E2 -972.094} C_VEL
LIN {X 0,Y 594.354,Z 249.07,A -85,B 0,C 180,E1 -974.218,E2 -974.218} C_VEL
LIN {X 0,Y 594.361,Z 249.069,A -85,B 0,C 180,E1 -976.32,E2 -976.32} C_VEL
LIN {X 0,Y 594.379,Z 249.068,A -85,B 0,C 180,E1 -979.094,E2 -979.094} C_VEL
LIN {X 0,Y 594.402,Z 249.069,A -85,B 0,C 180,E1 -981.842,E2 -981.842} C_VEL
LIN {X 0,Y 594.376,Z 249.066,A -85,B 0,C 180,E1 -984.571,E2 -984.571} C_VEL
LIN {X 0,Y 594.409,Z 249.067,A -85,B 0,C 180,E1 -987.288,E2 -987.288} C_VEL
LIN {X 0,Y 594.391,Z 249.067,A -85,B 0,C 180,E1 -989.999,E2 -989.999} C_VEL
LIN {X 0,Y 594.392,Z 249.064,A -85,B 0,C 180,E1 -992.71,E2 -992.71} C_VEL
LIN {X 0,Y 594.39,Z 249.073,A -85,B 0,C 180,E1 -995.427,E2 -995.427} C_VEL
LIN {X 0,Y 594.368,Z 249.068,A -85,B 0,C 180,E1 -998.156,E2 -998.156} C_VEL
LIN {X 0,Y 594.379,Z 249.069,A -85,B 0,C 180,E1 -1001.074,E2 -1001.074} C_VEL
LIN {X 0,Y 594.367,Z 249.074,A -85,B 0,C 180,E1 -1003.678,E2 -1003.678} C_VEL
LIN {X 0,Y 594.376,Z 249.066,A -85,B 0,C 180,E1 -1006.717,E2 -1006.717} C_VEL
LIN {X 0,Y 594.357,Z 249.077,A -85,B 0,C 180,E1 -1009.334,E2 -1009.334} C_VEL
LIN {X 0,Y 594.358,Z 249.077,A -85,B 0,C 180,E1 -1011.502,E2 -1011.502} C_VEL
LIN {X 0,Y 594.375,Z 249.066,A -85,B 0,C 180,E1 -1014.445,E2 -1014.445} C_VEL
LIN {X 0,Y 594.376,Z 249.067,A -85,B 0,C 180,E1 -1016.699,E2 -1016.699} C_VEL
LIN {X 0,Y 594.368,Z 249.071,A -85,B 0,C 180,E1 -1018.998,E2 -1018.998} C_VEL
LIN {X 0,Y 594.377,Z 249.071,A -85,B 0,C 180,E1 -1021.644,E2 -1021.644} C_VEL
LIN {X 0,Y 594.39,Z 249.065,A -85,B 0,C 180,E1 -1024.578,E2 -1024.578} C_VEL
LIN {X 0,Y 594.375,Z 249.072,A -85,B 0,C 180,E1 -1027.608,E2 -1027.608} C_VEL
LIN {X 0,Y 594.355,Z 249.069,A -85,B 0,C 180,E1 -1030.566,E2 -1030.566} C_VEL
LIN {X 0,Y 594.365,Z 249.078,A -85,B 0,C 180,E1 -1033.298,E2 -1033.298} C_VEL
LIN {X 0,Y 594.367,Z 249.067,A -85,B 0,C 180,E1 -1036.159,E2 -1036.159} C_VEL
LIN {X 0,Y 594.368,Z 249.076,A -85,B 0,C 180,E1 -1039.177,E2 -1039.177} C_VEL
LIN {X 0,Y 594.367,Z 249.067,A -85,B 0,C 180,E1 -1042.059,E2 -1042.059} C_VEL
LIN {X 0,Y 594.371,Z 249.069,A -85,B 0,C 180,E1 -1044.671,E2 -1044.671} C_VEL
LIN {X 0,Y 594.364,Z 249.076,A -85,B 0,C 180,E1 -1047.088,E2 -1047.088} C_VEL
LIN {X 0,Y 594.371,Z 249.069,A -85,B 0,C 180,E1 -1049.672,E2 -1049.672} C_VEL
LIN {X 0,Y 594.358,Z 249.069,A -85,B 0,C 180,E1 -1052.539,E2 -1052.539} C_VEL
LIN {X 0,Y 594.363,Z 249.072,A -85,B 0,C 180,E1 -1054.807,E2 -1054.807} C_VEL
LIN {X 0,Y 594.351,Z 249.078,A -85,B 0,C 180,E1 -1057.264,E2 -1057.264} C_VEL
LIN {X 0,Y 594.359,Z 249.068,A -85,B 0,C 180,E1 -1059.946,E2 -1059.946} C_VEL
LIN {X 0,Y 594.378,Z 249.071,A -85,B 0,C 180,E1 -1062.807,E2 -1062.807} C_VEL
LIN {X 0,Y 594.361,Z 249.068,A -85,B 0,C 180,E1 -1065.831,E2 -1065.831} C_VEL
LIN {X 0,Y 594.381,Z 249.066,A -85,B 0,C 180,E1 -1068.405,E2 -1068.405} C_VEL
LIN {X 0,Y 594.368,Z 249.076,A -85,B 0,C 180,E1 -1071.158,E2 -1071.158} C_VEL
LIN {X 0,Y 594.383,Z 249.071,A -85,B 0,C 180,E1 -1073.31,E2 -1073.31} C_VEL
LIN {X 0,Y 594.331,Z 249.071,A -85,B 0,C 180,E1 -1075.932,E2 -1075.932} C_VEL
LIN {X 0,Y 594.37,Z 249.066,A -85,B 0,C 180,E1 -1077.968,E2 -1077.968} C_VEL
LIN {X 0,Y 594.422,Z 249.065,A -85,B 0,C 180,E1 -1080.678,E2 -1080.678} C_VEL
LIN {X 0,Y 594.363,Z 249.071,A -85,B 0,C 180,E1 -1083.39,E2 -1083.39} C_VEL
LIN {X 0,Y 594.374,Z 249.069,A -85,B 0,C 180,E1 -1085.428,E2 -1085.428} C_VEL
LIN {X 0,Y 594.399,Z 249.063,A -85,B 0,C 180,E1 -1088.157,E2 -1088.157} C_VEL
LIN {X 0,Y 594.388,Z 249.073,A -85,B 0,C 180,E1 -1091.081,E2 -1091.081} C_VEL
LIN {X 0,Y 594.376,Z 249.066,A -85,B 0,C 180,E1 -1094.174,E2 -1094.174} C_VEL
LIN {X 0,Y 594.376,Z 249.072,A -85,B 0,C 180,E1 -1097.194,E2 -1097.194} C_VEL
LIN {X 0,Y 594.363,Z 249.068,A -85,B 0,C 180,E1 -1100.055,E2 -1100.055} C_VEL
LIN {X 0,Y 594.356,Z 249.077,A -85,B 0,C 180,E1 -1102.968,E2 -1102.968} C_VEL
LIN {X 0,Y 594.351,Z 249.074,A -85,B 0,C 180,E1 -1105.195,E2 -1105.195} C_VEL
LIN {X 0,Y 594.356,Z 249.069,A -85,B 0,C 180,E1 -1107.524,E2 -1107.524} C_VEL
LIN {X 0,Y 594.375,Z 249.068,A -85,B 0,C 180,E1 -1110.329,E2 -1110.329} C_VEL
LIN {X 0,Y 594.368,Z 249.075,A -85,B 0,C 180,E1 -1112.951,E2 -1112.951} C_VEL
LIN {X 0,Y 594.342,Z 249.072,A -85,B 0,C 180,E1 -1115.41,E2 -1115.41} C_VEL
LIN {X 0,Y 594.376,Z 249.066,A -85,B 0,C 180,E1 -1117.942,E2 -1117.942} C_VEL
LIN {X 0,Y 594.365,Z 249.077,A -85,B 0,C 180,E1 -1120.823,E2 -1120.823} C_VEL
LIN {X 0,Y 594.344,Z 249.072,A -85,B 0,C 180,E1 -1123.302,E2 -1123.302} C_VEL
LIN {X 0,Y 594.367,Z 249.069,A -85,B 0,C 180,E1 -1126.161,E2 -1126.161} C_VEL
LIN {X 0,Y 594.365,Z 249.071,A -85,B 0,C 180,E1 -1129.18,E2 -1129.18} C_VEL
LIN {X 0,Y 594.373,Z 249.068,A -85,B 0,C 180,E1 -1132.06,E2 -1132.06} C_VEL
LIN {X 0,Y 594.344,Z 249.08,A -85,B 0,C 180,E1 -1134.678,E2 -1134.678} C_VEL
LIN {X 0,Y 594.368,Z 249.071,A -85,B 0,C 180,E1 -1137.09,E2 -1137.09} C_VEL
LIN {X 0,Y 594.364,Z 249.068,A -85,B 0,C 180,E1 -1139.676,E2 -1139.676} C_VEL
LIN {X 0,Y 594.37,Z 249.077,A -85,B 0,C 180,E1 -1142.54,E2 -1142.54} C_VEL
LIN {X 0,Y 594.384,Z 249.081,A -85,B 0,C 180,E1 -1143.088,E2 -1143.088} C_VEL
LIN {X 0,Y 595.219,Z 253.922,A -85,B 0,C 180,E1 -1143.679,E2 -1143.679} C_VEL
LIN {X 0,Y 595.032,Z 279.279,A -85,B 0,C 180,E1 -1146.509,E2 -1146.509} C_VEL
LIN {X 0,Y 594.858,Z 305.935,A -85,B 0,C 180,E1 -1149.423,E2 -1149.423} C_VEL
LIN {X 0,Y 594.769,Z 321.631,A -85,B 0,C 180,E1 -1151.098,E2 -1151.098} C_VEL
LIN {X 0,Y 595.313,Z 325.039,A -85,B 0,C 180,E1 -1151.158,E2 -1151.158} C_VEL
LIN {X 0,Y 595.093,Z 488.156,A -85,B 0,C 180,E1 -1153.195,E2 -1153.195} C_VEL
LIN {X 0,Y 595.025,Z 503.752,A -85,B 0,C 180,E1 -1153.534,E2 -1153.534} C_VEL
LIN {X 0,Y 594.932,Z 519.076,A -85,B 0,C 180,E1 -1154.016,E2 -1154.016} C_VEL
LIN {X 0,Y 594.857,Z 532.788,A -85,B 0,C 180,E1 -1154.585,E2 -1154.585} C_VEL
LIN {X 0,Y 594.736,Z 546.256,A -85,B 0,C 180,E1 -1155.283,E2 -1155.283} C_VEL
LIN {X 0,Y 594.679,Z 558.809,A -85,B 0,C 180,E1 -1156.076,E2 -1156.076} C_VEL
LIN {X 0,Y 594.56,Z 571.299,A -85,B 0,C 180,E1 -1157.022,E2 -1157.022} C_VEL
LIN {X 0,Y 594.464,Z 582.759,A -85,B 0,C 180,E1 -1158.061,E2 -1158.061} C_VEL
LIN {X 0,Y 594.389,Z 592.398,A -85,B 0,C 180,E1 -1159.096,E2 -1159.096} C_VEL
LIN {X 0,Y 594.366,Z 601.863,A -85,B 0,C 180,E1 -1160.301,E2 -1160.301} C_VEL
LIN {X 0,Y 594.31,Z 609.737,A -85,B 0,C 180,E1 -1161.501,E2 -1161.501} C_VEL
LIN {X 0,Y 594.292,Z 617.093,A -85,B 0,C 180,E1 -1162.868,E2 -1162.868} C_VEL
LIN {X 0,Y 594.296,Z 622.928,A -85,B 0,C 180,E1 -1164.232,E2 -1164.232} C_VEL
LIN {X 0,Y 594.232,Z 626.387,A -85,B 0,C 180,E1 -1165.252,E2 -1165.252} C_VEL
LIN {X 0,Y 594.256,Z 629.889,A -85,B 0,C 180,E1 -1166.611,E2 -1166.611} C_VEL
LIN {X 0,Y 594.24,Z 632.194,A -85,B 0,C 180,E1 -1167.968,E2 -1167.968} C_VEL
LIN {X 0,Y 594.237,Z 633.35,A -85,B 0,C 180,E1 -1169.323,E2 -1169.323} C_VEL
LIN {X 0,Y 594.237,Z 633.35,A -85,B 0,C 180,E1 -1170.679,E2 -1170.679} C_VEL
LIN {X 0,Y 594.24,Z 632.191,A -85,B 0,C 180,E1 -1172.034,E2 -1172.034} C_VEL
LIN {X 0,Y 594.256,Z 629.884,A -85,B 0,C 180,E1 -1173.391,E2 -1173.391} C_VEL
LIN {X 0,Y 594.232,Z 626.381,A -85,B 0,C 180,E1 -1174.75,E2 -1174.75} C_VEL
LIN {X 0,Y 594.275,Z 621.604,A -85,B 0,C 180,E1 -1176.111,E2 -1176.111} C_VEL
LIN {X 0,Y 594.288,Z 615.42,A -85,B 0,C 180,E1 -1177.475,E2 -1177.475} C_VEL
LIN {X 0,Y 594.331,Z 607.646,A -85,B 0,C 180,E1 -1178.844,E2 -1178.844} C_VEL
LIN {X 0,Y 594.387,Z 599.363,A -85,B 0,C 180,E1 -1180.045,E2 -1180.045} C_VEL
LIN {X 0,Y 594.435,Z 589.555,A -85,B 0,C 180,E1 -1181.232,E2 -1181.232} C_VEL
LIN {X 0,Y 594.531,Z 579.183,A -85,B 0,C 180,E1 -1182.286,E2 -1182.286} C_VEL
LIN {X 0,Y 594.582,Z 567.006,A -85,B 0,C 180,E1 -1183.327,E2 -1183.327} C_VEL
LIN {X 0,Y 594.697,Z 555.062,A -85,B 0,C 180,E1 -1184.178,E2 -1184.178} C_VEL
LIN {X 0,Y 594.783,Z 541.509,A -85,B 0,C 180,E1 -1184.98,E2 -1184.98} C_VEL
LIN {X 0,Y 594.906,Z 526.821,A -85,B 0,C 180,E1 -1185.679,E2 -1185.679} C_VEL
LIN {X 0,Y 594.968,Z 512.594,A -85,B 0,C 180,E1 -1186.205,E2 -1186.205} C_VEL
LIN {X 0,Y 595.05,Z 498.083,A -85,B 0,C 180,E1 -1186.604,E2 -1186.604} C_VEL
LIN {X 0,Y 595.071,Z 482.649,A -85,B 0,C 180,E1 -1186.887,E2 -1186.887} C_VEL
LIN {X 0,Y 595.236,Z 324.22,A -85,B 0,C 180,E1 -1188.854,E2 -1188.854} C_VEL
LIN {X 0,Y 594.743,Z 321.448,A -85,B 0,C 180,E1 -1188.907,E2 -1188.907} C_VEL
LIN {X 0,Y 594.889,Z 295.921,A -85,B 0,C 180,E1 -1191.666,E2 -1191.666} C_VEL
LIN {X 0,Y 595.077,Z 270.93,A -85,B 0,C 180,E1 -1194.417,E2 -1194.417} C_VEL
LIN {X 0,Y 595.223,Z 253.638,A -85,B 0,C 180,E1 -1196.353,E2 -1196.353} C_VEL
LIN {X 0,Y 594.365,Z 249.076,A -85,B 0,C 180,E1 -1196.938,E2 -1196.938} C_VEL
LIN {X 0,Y 594.364,Z 249.071,A -85,B 0,C 180,E1 -1199.778,E2 -1199.778} C_VEL
LIN {X 0,Y 594.358,Z 249.069,A -85,B 0,C 180,E1 -1202.148,E2 -1202.148} C_VEL
LIN {X 0,Y 594.376,Z 249.069,A -85,B 0,C 180,E1 -1204.581,E2 -1204.581} C_VEL
LIN {X 0,Y 594.393,Z 249.067,A -85,B 0,C 180,E1 -1207.609,E2 -1207.609} C_VEL
LIN {X 0,Y 594.366,Z 249.072,A -85,B 0,C 180,E1 -1210.568,E2 -1210.568} C_VEL
LIN {X 0,Y 594.37,Z 249.071,A -85,B 0,C 180,E1 -1213.3,E2 -1213.3} C_VEL
LIN {X 0,Y 594.373,Z 249.068,A -85,B 0,C 180,E1 -1216.161,E2 -1216.161} C_VEL
LIN {X 0,Y 594.383,Z 249.073,A -85,B 0,C 180,E1 -1218.536,E2 -1218.536} C_VEL
LIN {X 0,Y 594.377,Z 249.068,A -85,B 0,C 180,E1 -1221.297,E2 -1221.297} C_VEL
LIN {X 0,Y 594.354,Z 249.07,A -85,B 0,C 180,E1 -1223.755,E2 -1223.755} C_VEL
LIN {X 0,Y 594.384,Z 249.072,A -85,B 0,C 180,E1 -1226.239,E2 -1226.239} C_VEL
LIN {X 0,Y 594.372,Z 249.074,A -85,B 0,C 180,E1 -1228.65,E2 -1228.65} C_VEL
LIN {X 0,Y 594.383,Z 249.067,A -85,B 0,C 180,E1 -1231.043,E2 -1231.043} C_VEL
LIN {X 0,Y 594.393,Z 249.07,A -85,B 0,C 180,E1 -1233.977,E2 -1233.977} C_VEL
LIN {X 0,Y 594.377,Z 249.076,A -85,B 0,C 180,E1 -1236.295,E2 -1236.295} C_VEL
LIN {X 0,Y 594.4,Z 249.184,A -85,B 0,C 180,E1 -1239.079,E2 -1239.079} C_VEL
LIN {X 0,Y 594.632,Z 255.152,A -85,B 0,C 180,E1 -1239.955,E2 -1239.955} C_VEL
LIN {X 0,Y 594.588,Z 263.514,A -85,B 0,C 180,E1 -1241.16,E2 -1241.16} C_VEL
LIN {X 0,Y 595.328,Z 267.566,A -85,B 0,C 180,E1 -1241.235,E2 -1241.235} C_VEL
LIN {X 0,Y 595.096,Z 428.329,A -85,B 0,C 180,E1 -1243.244,E2 -1243.244} C_VEL
LIN {X 0,Y 594.998,Z 444.393,A -85,B 0,C 180,E1 -1243.598,E2 -1243.598} C_VEL
LIN {X 0,Y 594.959,Z 458.988,A -85,B 0,C 180,E1 -1244.059,E2 -1244.059} C_VEL
LIN {X 0,Y 594.82,Z 473.649,A -85,B 0,C 180,E1 -1244.67,E2 -1244.67} C_VEL
LIN {X 0,Y 594.732,Z 486.961,A -85,B 0,C 180,E1 -1245.369,E2 -1245.369} C_VEL
LIN {X 0,Y 594.67,Z 499.995,A -85,B 0,C 180,E1 -1246.201,E2 -1246.201} C_VEL
LIN {X 0,Y 594.553,Z 512.832,A -85,B 0,C 180,E1 -1247.194,E2 -1247.194} C_VEL
LIN {X 0,Y 594.469,Z 524.054,A -85,B 0,C 180,E1 -1248.232,E2 -1248.232} C_VEL
LIN {X 0,Y 594.414,Z 534.943,A -85,B 0,C 180,E1 -1249.44,E2 -1249.44} C_VEL
LIN {X 0,Y 594.332,Z 543.976,A -85,B 0,C 180,E1 -1250.642,E2 -1250.642} C_VEL
LIN {X 0,Y 594.312,Z 551.477,A -85,B 0,C 180,E1 -1251.841,E2 -1251.841} C_VEL
LIN {X 0,Y 594.278,Z 558.496,A -85,B 0,C 180,E1 -1253.208,E2 -1253.208} C_VEL
LIN {X 0,Y 594.272,Z 563.995,A -85,B 0,C 180,E1 -1254.571,E2 -1254.571} C_VEL
LIN {X 0,Y 594.25,Z 568.176,A -85,B 0,C 180,E1 -1255.93,E2 -1255.93} C_VEL
LIN {X 0,Y 594.221,Z 571.107,A -85,B 0,C 180,E1 -1257.288,E2 -1257.288} C_VEL
LIN {X 0,Y 594.247,Z 572.883,A -85,B 0,C 180,E1 -1258.644,E2 -1258.644} C_VEL
LIN {X 0,Y 594.232,Z 573.496,A -85,B 0,C 180,E1 -1259.999,E2 -1259.999} C_VEL
LIN {X 0,Y 594.245,Z 572.95,A -85,B 0,C 180,E1 -1261.355,E2 -1261.355} C_VEL
LIN {X 0,Y 594.224,Z 571.256,A -85,B 0,C 180,E1 -1262.711,E2 -1262.711} C_VEL
LIN {X 0,Y 594.252,Z 568.414,A -85,B 0,C 180,E1 -1264.069,E2 -1264.069} C_VEL
LIN {X 0,Y 594.272,Z 564.323,A -85,B 0,C 180,E1 -1265.428,E2 -1265.428} C_VEL
LIN {X 0,Y 594.277,Z 558.923,A -85,B 0,C 180,E1 -1266.791,E2 -1266.791} C_VEL
LIN {X 0,Y 594.312,Z 552.008,A -85,B 0,C 180,E1 -1268.157,E2 -1268.157} C_VEL
LIN {X 0,Y 594.327,Z 544.58,A -85,B 0,C 180,E1 -1269.357,E2 -1269.357} C_VEL
LIN {X 0,Y 594.414,Z 535.669,A -85,B 0,C 180,E1 -1270.559,E2 -1270.559} C_VEL
LIN {X 0,Y 594.43,Z 526.572,A -85,B 0,C 180,E1 -1271.594,E2 -1271.594} C_VEL
LIN {X 0,Y 594.512,Z 515.853,A -85,B 0,C 180,E1 -1272.632,E2 -1272.632} C_VEL
LIN {X 0,Y 594.595,Z 504.378,A -85,B 0,C 180,E1 -1273.569,E2 -1273.569} C_VEL
LIN {X 0,Y 593.955,Z 499.776,A -85,B 0,C 180,E1 -1273.921,E2 -1273.921} C_VEL
LIN {X 0,Y 591.199,Z 492.28,A -85,B 0,C 180,E1 -1274.494,E2 -1274.494} C_VEL
LIN {X 0,Y 588.481,Z 484.5,A -85,B 0,C 180,E1 -1275.027,E2 -1275.027} C_VEL
LIN {X 0,Y 587.892,Z 479.431,A -85,B 0,C 180,E1 -1275.315,E2 -1275.315} C_VEL
LIN {X 0,Y 588.056,Z 465.755,A -85,B 0,C 180,E1 -1275.954,E2 -1275.954} C_VEL
LIN {X 0,Y 588.178,Z 451.327,A -85,B 0,C 180,E1 -1276.485,E2 -1276.485} C_VEL
LIN {X 0,Y 588.236,Z 435.558,A -85,B 0,C 180,E1 -1276.904,E2 -1276.904} C_VEL
LIN {X 0,Y 588.32,Z 419.3,A -85,B 0,C 180,E1 -1277.178,E2 -1277.178} C_VEL
LIN {X 0,Y 588.566,Z 268.326,A -85,B 0,C 180,E1 -1279.069,E2 -1279.069} C_VEL
LIN {X 0,Y 587.625,Z 263.347,A -85,B 0,C 180,E1 -1279.186,E2 -1279.186} C_VEL
LIN {X 0,Y 587.683,Z 252.042,A -85,B 0,C 180,E1 -1280.84,E2 -1280.84} C_VEL
LIN {X 0,Y 587.339,Z 249.949,A -85,B 0,C 180,E1 -1281.181,E2 -1281.181} C_VEL
LIN {X 0,Y 587.306,Z 249.957,A -85,B 0,C 180,E1 -1284.007,E2 -1284.007} C_VEL
LIN {X 0,Y 587.309,Z 249.951,A -85,B 0,C 180,E1 -1286.279,E2 -1286.279} C_VEL
LIN {X 0,Y 587.343,Z 249.943,A -85,B 0,C 180,E1 -1289.131,E2 -1289.131} C_VEL
LIN {X 0,Y 587.338,Z 249.952,A -85,B 0,C 180,E1 -1291.834,E2 -1291.834} C_VEL
LIN {X 0,Y 587.34,Z 249.945,A -85,B 0,C 180,E1 -1294.346,E2 -1294.346} C_VEL
LIN {X 0,Y 587.341,Z 249.948,A -85,B 0,C 180,E1 -1297.607,E2 -1297.607} C_VEL
LIN {X 0,Y 587.306,Z 249.95,A -85,B 0,C 180,E1 -1300.254,E2 -1300.254} C_VEL
LIN {X 0,Y 587.31,Z 249.947,A -85,B 0,C 180,E1 -1303.117,E2 -1303.117} C_VEL
LIN {X 0,Y 587.307,Z 249.953,A -85,B 0,C 180,E1 -1306.047,E2 -1306.047} C_VEL
LIN {X 0,Y 587.33,Z 249.944,A -85,B 0,C 180,E1 -1308.924,E2 -1308.924} C_VEL
LIN {X 0,Y 587.325,Z 249.95,A -85,B 0,C 180,E1 -1311.52,E2 -1311.52} C_VEL
LIN {X 0,Y 587.289,Z 249.954,A -85,B 0,C 180,E1 -1314.099,E2 -1314.099} C_VEL
LIN {X 0,Y 587.323,Z 249.944,A -85,B 0,C 180,E1 -1316.602,E2 -1316.602} C_VEL
LIN {X 0,Y 587.331,Z 249.949,A -85,B 0,C 180,E1 -1319.489,E2 -1319.489} C_VEL
LIN {X 0,Y 587.303,Z 249.95,A -85,B 0,C 180,E1 -1322.179,E2 -1322.179} C_VEL
LIN {X 0,Y 587.316,Z 249.946,A -85,B 0,C 180,E1 -1324.482,E2 -1324.482} C_VEL
LIN {X 0,Y 587.332,Z 249.95,A -85,B 0,C 180,E1 -1327.485,E2 -1327.485} C_VEL
LIN {X 0,Y 587.305,Z 249.947,A -85,B 0,C 180,E1 -1330.423,E2 -1330.423} C_VEL
LIN {X 0,Y 587.351,Z 249.946,A -85,B 0,C 180,E1 -1333.31,E2 -1333.31} C_VEL
LIN {X 0,Y 587.34,Z 249.945,A -85,B 0,C 180,E1 -1336.153,E2 -1336.153} C_VEL
LIN {X 0,Y 587.342,Z 249.943,A -85,B 0,C 180,E1 -1338.962,E2 -1338.962} C_VEL
LIN {X 0,Y 587.358,Z 249.948,A -85,B 0,C 180,E1 -1341.744,E2 -1341.744} C_VEL
LIN {X 0,Y 587.341,Z 249.942,A -85,B 0,C 180,E1 -1344.506,E2 -1344.506} C_VEL
LIN {X 0,Y 587.374,Z 249.943,A -85,B 0,C 180,E1 -1347.256,E2 -1347.256} C_VEL
LIN {X 0,Y 587.361,Z 249.943,A -85,B 0,C 180,E1 -1349.999,E2 -1349.999} C_VEL
LIN {X 0,Y 587.36,Z 249.94,A -85,B 0,C 180,E1 -1352.742,E2 -1352.742} C_VEL
LIN {X 0,Y 587.352,Z 249.951,A -85,B 0,C 180,E1 -1355.492,E2 -1355.492} C_VEL
LIN {X 0,Y 587.329,Z 249.944,A -85,B 0,C 180,E1 -1358.255,E2 -1358.255} C_VEL
LIN {X 0,Y 587.337,Z 249.947,A -85,B 0,C 180,E1 -1361.133,E2 -1361.133} C_VEL
LIN {X 0,Y 587.345,Z 249.942,A -85,B 0,C 180,E1 -1364.256,E2 -1364.256} C_VEL
LIN {X 0,Y 587.338,Z 249.952,A -85,B 0,C 180,E1 -1367.405,E2 -1367.405} C_VEL
LIN {X 0,Y 587.315,Z 249.945,A -85,B 0,C 180,E1 -1370.304,E2 -1370.304} C_VEL
LIN {X 0,Y 587.308,Z 249.954,A -85,B 0,C 180,E1 -1373.258,E2 -1373.258} C_VEL
LIN {X 0,Y 587.32,Z 249.953,A -85,B 0,C 180,E1 -1375.516,E2 -1375.516} C_VEL
LIN {X 0,Y 587.332,Z 249.947,A -85,B 0,C 180,E1 -1377.817,E2 -1377.817} C_VEL
LIN {X 0,Y 587.329,Z 249.944,A -85,B 0,C 180,E1 -1380.51,E2 -1380.51} C_VEL
LIN {X 0,Y 587.321,Z 249.955,A -85,B 0,C 180,E1 -1383.396,E2 -1383.396} C_VEL
LIN {X 0,Y 587.289,Z 249.951,A -85,B 0,C 180,E1 -1385.899,E2 -1385.899} C_VEL
LIN {X 0,Y 587.317,Z 249.945,A -85,B 0,C 180,E1 -1388.479,E2 -1388.479} C_VEL
LIN {X 0,Y 587.324,Z 249.952,A -85,B 0,C 180,E1 -1391.156,E2 -1391.156} C_VEL
LIN {X 0,Y 587.319,Z 249.945,A -85,B 0,C 180,E1 -1394.114,E2 -1394.114} C_VEL
LIN {X 0,Y 587.308,Z 249.952,A -85,B 0,C 180,E1 -1396.994,E2 -1396.994} C_VEL
LIN {X 0,Y 587.303,Z 249.95,A -85,B 0,C 180,E1 -1399.746,E2 -1399.746} C_VEL
LIN {X 0,Y 587.33,Z 249.944,A -85,B 0,C 180,E1 -1402.392,E2 -1402.392} C_VEL
LIN {X 0,Y 587.338,Z 249.948,A -85,B 0,C 180,E1 -1404.946,E2 -1404.946} C_VEL
LIN {X 0,Y 587.324,Z 249.951,A -85,B 0,C 180,E1 -1407.421,E2 -1407.421} C_VEL
LIN {X 0,Y 587.318,Z 249.946,A -85,B 0,C 180,E1 -1409.83,E2 -1409.83} C_VEL
LIN {X 0,Y 587.335,Z 249.943,A -85,B 0,C 180,E1 -1412.307,E2 -1412.307} C_VEL
LIN {X 0,Y 587.336,Z 249.952,A -85,B 0,C 180,E1 -1415.242,E2 -1415.242} C_VEL
LIN {X 0,Y 587.308,Z 249.946,A -85,B 0,C 180,E1 -1418.226,E2 -1418.226} C_VEL
LIN {X 0,Y 587.335,Z 249.953,A -85,B 0,C 180,E1 -1421.151,E2 -1421.151} C_VEL
LIN {X 0,Y 587.308,Z 249.946,A -85,B 0,C 180,E1 -1424.025,E2 -1424.025} C_VEL
LIN {X 0,Y 587.339,Z 249.942,A -85,B 0,C 180,E1 -1426.154,E2 -1426.154} C_VEL
LIN {X 0,Y 587.33,Z 249.952,A -85,B 0,C 180,E1 -1428.963,E2 -1428.963} C_VEL
LIN {X 0,Y 587.326,Z 249.945,A -85,B 0,C 180,E1 -1431.745,E2 -1431.745} C_VEL
LIN {X 0,Y 587.351,Z 249.943,A -85,B 0,C 180,E1 -1434.508,E2 -1434.508} C_VEL
LIN {X 0,Y 587.359,Z 249.947,A -85,B 0,C 180,E1 -1437.257,E2 -1437.257} C_VEL
LIN {X 0,Y 587.358,Z 249.94,A -85,B 0,C 180,E1 -1440.001,E2 -1440.001} C_VEL
LIN {X 0,Y 587.373,Z 249.944,A -85,B 0,C 180,E1 -1442.744,E2 -1442.744} C_VEL
LIN {X 0,Y 587.338,Z 249.945,A -85,B 0,C 180,E1 -1445.494,E2 -1445.494} C_VEL
LIN {X 0,Y 587.354,Z 249.941,A -85,B 0,C 180,E1 -1448.256,E2 -1448.256} C_VEL
LIN {X 0,Y 587.351,Z 249.948,A -85,B 0,C 180,E1 -1451.142,E2 -1451.142} C_VEL
LIN {X 0,Y 587.352,Z 249.942,A -85,B 0,C 180,E1 -1454.261,E2 -1454.261} C_VEL
LIN {X 0,Y 587.336,Z 249.946,A -85,B 0,C 180,E1 -1457.407,E2 -1457.407} C_VEL
LIN {X 0,Y 587.301,Z 249.948,A -85,B 0,C 180,E1 -1459.577,E2 -1459.577} C_VEL
LIN {X 0,Y 587.313,Z 249.946,A -85,B 0,C 180,E1 -1461.775,E2 -1461.775} C_VEL
LIN {X 0,Y 587.336,Z 249.951,A -85,B 0,C 180,E1 -1464.76,E2 -1464.76} C_VEL
LIN {X 0,Y 587.331,Z 249.944,A -85,B 0,C 180,E1 -1467.692,E2 -1467.692} C_VEL
LIN {X 0,Y 587.326,Z 249.949,A -85,B 0,C 180,E1 -1470.511,E2 -1470.511} C_VEL
LIN {X 0,Y 587.318,Z 249.947,A -85,B 0,C 180,E1 -1473.398,E2 -1473.398} C_VEL
LIN {X 0,Y 587.282,Z 249.949,A -85,B 0,C 180,E1 -1475.901,E2 -1475.901} C_VEL
LIN {X 0,Y 587.32,Z 249.95,A -85,B 0,C 180,E1 -1478.48,E2 -1478.48} C_VEL
LIN {X 0,Y 587.324,Z 249.948,A -85,B 0,C 180,E1 -1481.158,E2 -1481.158} C_VEL
LIN {X 0,Y 587.309,Z 249.947,A -85,B 0,C 180,E1 -1484.114,E2 -1484.114} C_VEL
LIN {X 0,Y 587.299,Z 249.953,A -85,B 0,C 180,E1 -1486.994,E2 -1486.994} C_VEL
LIN {X 0,Y 587.306,Z 249.947,A -85,B 0,C 180,E1 -1489.747,E2 -1489.747} C_VEL
LIN {X 0,Y 587.336,Z 249.948,A -85,B 0,C 180,E1 -1492.393,E2 -1492.393} C_VEL
LIN {X 0,Y 587.349,Z 249.941,A -85,B 0,C 180,E1 -1495.781,E2 -1495.781} C_VEL
LIN {X 0,Y 587.341,Z 249.946,A -85,B 0,C 180,E1 -1498.233,E2 -1498.233} C_VEL
LIN {X 0,Y 587.339,Z 249.952,A -85,B 0,C 180,E1 -1500.869,E2 -1500.869} C_VEL
LIN {X 0,Y 587.387,Z 250.111,A -85,B 0,C 180,E1 -1502.862,E2 -1502.862} C_VEL
LIN {X 0,Y 588.467,Z 256.08,A -85,B 0,C 180,E1 -1503.601,E2 -1503.601} C_VEL
LIN {X 0,Y 588.209,Z 280.945,A -85,B 0,C 180,E1 -1506.407,E2 -1506.407} C_VEL
LIN {X 0,Y 587.978,Z 307.601,A -85,B 0,C 180,E1 -1509.354,E2 -1509.354} C_VEL
LIN {X 0,Y 587.852,Z 321.375,A -85,B 0,C 180,E1 -1510.855,E2 -1510.855} C_VEL
LIN {X 0,Y 588.613,Z 326.849,A -85,B 0,C 180,E1 -1510.959,E2 -1510.959} C_VEL
LIN {X 0,Y 588.307,Z 488.256,A -85,B 0,C 180,E1 -1512.997,E2 -1512.997} C_VEL
LIN {X 0,Y 588.226,Z 503.75,A -85,B 0,C 180,E1 -1513.338,E2 -1513.338} C_VEL
LIN {X 0,Y 588.07,Z 519.074,A -85,B 0,C 180,E1 -1513.824,E2 -1513.824} C_VEL
LIN {X 0,Y 587.988,Z 532.791,A -85,B 0,C 180,E1 -1514.4,E2 -1514.4} C_VEL
LIN {X 0,Y 587.835,Z 546.259,A -85,B 0,C 180,E1 -1515.106,E2 -1515.106} C_VEL
LIN {X 0,Y 587.738,Z 559.13,A -85,B 0,C 180,E1 -1515.931,E2 -1515.931} C_VEL
LIN {X 0,Y 587.583,Z 571.301,A -85,B 0,C 180,E1 -1516.866,E2 -1516.866} C_VEL
LIN {X 0,Y 587.453,Z 582.76,A -85,B 0,C 180,E1 -1517.916,E2 -1517.916} C_VEL
LIN {X 0,Y 587.348,Z 592.399,A -85,B 0,C 180,E1 -1518.964,E2 -1518.964} C_VEL
LIN {X 0,Y 587.304,Z 601.864,A -85,B 0,C 180,E1 -1520.183,E2 -1520.183} C_VEL
LIN {X 0,Y 587.264,Z 609.738,A -85,B 0,C 180,E1 -1521.398,E2 -1521.398} C_VEL
LIN {X 0,Y 587.215,Z 617.093,A -85,B 0,C 180,E1 -1522.782,E2 -1522.782} C_VEL
LIN {X 0,Y 587.224,Z 622.927,A -85,B 0,C 180,E1 -1524.162,E2 -1524.162} C_VEL
LIN {X 0,Y 587.136,Z 626.387,A -85,B 0,C 180,E1 -1525.195,E2 -1525.195} C_VEL
LIN {X 0,Y 587.179,Z 629.89,A -85,B 0,C 180,E1 -1526.57,E2 -1526.57} C_VEL
LIN {X 0,Y 587.138,Z 632.194,A -85,B 0,C 180,E1 -1527.943,E2 -1527.943} C_VEL
LIN {X 0,Y 587.137,Z 633.35,A -85,B 0,C 180,E1 -1529.315,E2 -1529.315} C_VEL
LIN {X 0,Y 587.137,Z 633.349,A -85,B 0,C 180,E1 -1530.687,E2 -1530.687} C_VEL
LIN {X 0,Y 587.138,Z 632.191,A -85,B 0,C 180,E1 -1532.059,E2 -1532.059} C_VEL
LIN {X 0,Y 587.179,Z 629.884,A -85,B 0,C 180,E1 -1533.432,E2 -1533.432} C_VEL
LIN {X 0,Y 587.136,Z 626.381,A -85,B 0,C 180,E1 -1534.807,E2 -1534.807} C_VEL
LIN {X 0,Y 587.178,Z 621.604,A -85,B 0,C 180,E1 -1536.185,E2 -1536.185} C_VEL
LIN {X 0,Y 587.231,Z 615.419,A -85,B 0,C 180,E1 -1537.566,E2 -1537.566} C_VEL
LIN {X 0,Y 587.267,Z 607.645,A -85,B 0,C 180,E1 -1538.951,E2 -1538.951} C_VEL
LIN {X 0,Y 587.351,Z 599.363,A -85,B 0,C 180,E1 -1540.166,E2 -1540.166} C_VEL
LIN {X 0,Y 587.401,Z 589.387,A -85,B 0,C 180,E1 -1541.386,E2 -1541.386} C_VEL
LIN {X 0,Y 587.522,Z 579.182,A -85,B 0,C 180,E1 -1542.435,E2 -1542.435} C_VEL
LIN {X 0,Y 587.629,Z 567.007,A -85,B 0,C 180,E1 -1543.487,E2 -1543.487} C_VEL
LIN {X 0,Y 587.777,Z 554.044,A -85,B 0,C 180,E1 -1544.417,E2 -1544.417} C_VEL
LIN {X 0,Y 587.889,Z 539.85,A -85,B 0,C 180,E1 -1545.249,E2 -1545.249} C_VEL
LIN {X 0,Y 588.052,Z 525.776,A -85,B 0,C 180,E1 -1545.911,E2 -1545.911} C_VEL
LIN {X 0,Y 588.172,Z 511.278,A -85,B 0,C 180,E1 -1546.442,E2 -1546.442} C_VEL
LIN {X 0,Y 588.282,Z 496.238,A -85,B 0,C 180,E1 -1546.845,E2 -1546.845} C_VEL
LIN {X 0,Y 588.325,Z 481.013,A -85,B 0,C 180,E1 -1547.111,E2 -1547.111} C_VEL
LIN {X 0,Y 588.487,Z 324.855,A -85,B 0,C 180,E1 -1549.071,E2 -1549.071} C_VEL
LIN {X 0,Y 587.835,Z 321.326,A -85,B 0,C 180,E1 -1549.151,E2 -1549.151} C_VEL
LIN {X 0,Y 588.051,Z 295.921,A -85,B 0,C 180,E1 -1551.931,E2 -1551.931} C_VEL
LIN {X 0,Y 588.339,Z 270.274,A -85,B 0,C 180,E1 -1554.789,E2 -1554.789} C_VEL
LIN {X 0,Y 588.469,Z 256.077,A -85,B 0,C 180,E1 -1556.4,E2 -1556.4} C_VEL
LIN {X 0,Y 587.362,Z 249.985,A -85,B 0,C 180,E1 -1557.153,E2 -1557.153} C_VEL
LIN {X 0,Y 587.319,Z 249.947,A -85,B 0,C 180,E1 -1560.172,E2 -1560.172} C_VEL
LIN {X 0,Y 587.335,Z 249.947,A -85,B 0,C 180,E1 -1562.58,E2 -1562.58} C_VEL
LIN {X 0,Y 587.325,Z 249.955,A -85,B 0,C 180,E1 -1565.056,E2 -1565.056} C_VEL
LIN {X 0,Y 587.341,Z 249.944,A -85,B 0,C 180,E1 -1567.838,E2 -1567.838} C_VEL
LIN {X 0,Y 587.319,Z 249.947,A -85,B 0,C 180,E1 -1570.255,E2 -1570.255} C_VEL
LIN {X 0,Y 587.318,Z 249.952,A -85,B 0,C 180,E1 -1573.118,E2 -1573.118} C_VEL
LIN {X 0,Y 587.329,Z 249.946,A -85,B 0,C 180,E1 -1576.05,E2 -1576.05} C_VEL
LIN {X 0,Y 587.339,Z 249.95,A -85,B 0,C 180,E1 -1578.925,E2 -1578.925} C_VEL
LIN {X 0,Y 587.326,Z 249.945,A -85,B 0,C 180,E1 -1581.52,E2 -1581.52} C_VEL
LIN {X 0,Y 587.294,Z 249.952,A -85,B 0,C 180,E1 -1584.1,E2 -1584.1} C_VEL
LIN {X 0,Y 587.34,Z 249.952,A -85,B 0,C 180,E1 -1586.603,E2 -1586.603} C_VEL
LIN {X 0,Y 587.339,Z 249.944,A -85,B 0,C 180,E1 -1589.491,E2 -1589.491} C_VEL
LIN {X 0,Y 587.311,Z 249.955,A -85,B 0,C 180,E1 -1592.18,E2 -1592.18} C_VEL
LIN {X 0,Y 587.333,Z 249.952,A -85,B 0,C 180,E1 -1594.483,E2 -1594.483} C_VEL
LIN {X 0,Y 587.341,Z 249.946,A -85,B 0,C 180,E1 -1597.486,E2 -1597.486} C_VEL
LIN {X 0,Y 587.365,Z 250.123,A -85,B 0,C 180,E1 -1598.955,E2 -1598.955} C_VEL
LIN {X 0,Y 587.73,Z 255.156,A -85,B 0,C 180,E1 -1599.709,E2 -1599.709} C_VEL
LIN {X 0,Y 587.614,Z 263.467,A -85,B 0,C 180,E1 -1600.921,E2 -1600.921} C_VEL
LIN {X 0,Y 588.621,Z 268.535,A -85,B 0,C 180,E1 -1601.025,E2 -1601.025} C_VEL
LIN {X 0,Y 588.297,Z 428.328,A -85,B 0,C 180,E1 -1603.045,E2 -1603.045} C_VEL
LIN {X 0,Y 588.194,Z 444.392,A -85,B 0,C 180,E1 -1603.402,E2 -1603.402} C_VEL
LIN {X 0,Y 588.104,Z 458.99,A -85,B 0,C 180,E1 -1603.868,E2 -1603.868} C_VEL
LIN {X 0,Y 587.972,Z 473.645,A -85,B 0,C 180,E1 -1604.487,E2 -1604.487} C_VEL
LIN {X 0,Y 587.846,Z 486.963,A -85,B 0,C 180,E1 -1605.193,E2 -1605.193} C_VEL
LIN {X 0,Y 587.737,Z 500.167,A -85,B 0,C 180,E1 -1606.047,E2 -1606.047} C_VEL
LIN {X 0,Y 587.559,Z 512.833,A -85,B 0,C 180,E1 -1607.039,E2 -1607.039} C_VEL
LIN {X 0,Y 587.448,Z 524.052,A -85,B 0,C 180,E1 -1608.09,E2 -1608.09} C_VEL
LIN {X 0,Y 587.384,Z 534.945,A -85,B 0,C 180,E1 -1609.312,E2 -1609.312} C_VEL
LIN {X 0,Y 587.279,Z 543.973,A -85,B 0,C 180,E1 -1610.529,E2 -1610.529} C_VEL
LIN {X 0,Y 587.254,Z 551.475,A -85,B 0,C 180,E1 -1611.743,E2 -1611.743} C_VEL
LIN {X 0,Y 587.21,Z 558.502,A -85,B 0,C 180,E1 -1613.126,E2 -1613.126} C_VEL
LIN {X 0,Y 587.197,Z 563.996,A -85,B 0,C 180,E1 -1614.505,E2 -1614.505} C_VEL
LIN {X 0,Y 587.166,Z 568.18,A -85,B 0,C 180,E1 -1615.881,E2 -1615.881} C_VEL
LIN {X 0,Y 587.127,Z 571.107,A -85,B 0,C 180,E1 -1617.255,E2 -1617.255} C_VEL
LIN {X 0,Y 587.146,Z 572.878,A -85,B 0,C 180,E1 -1618.628,E2 -1618.628} C_VEL
LIN {X 0,Y 587.133,Z 573.496,A -85,B 0,C 180,E1 -1619.999,E2 -1619.999} C_VEL
LIN {X 0,Y 587.145,Z 572.953,A -85,B 0,C 180,E1 -1621.371,E2 -1621.371} C_VEL
LIN {X 0,Y 587.13,Z 571.254,A -85,B 0,C 180,E1 -1622.744,E2 -1622.744} C_VEL
LIN {X 0,Y 587.168,Z 568.416,A -85,B 0,C 180,E1 -1624.118,E2 -1624.118} C_VEL
LIN {X 0,Y 587.197,Z 564.316,A -85,B 0,C 180,E1 -1625.494,E2 -1625.494} C_VEL
LIN {X 0,Y 587.209,Z 558.919,A -85,B 0,C 180,E1 -1626.873,E2 -1626.873} C_VEL
LIN {X 0,Y 587.251,Z 551.999,A -85,B 0,C 180,E1 -1628.256,E2 -1628.256} C_VEL
LIN {X 0,Y 587.275,Z 544.571,A -85,B 0,C 180,E1 -1629.47,E2 -1629.47} C_VEL
LIN {X 0,Y 587.384,Z 535.669,A -85,B 0,C 180,E1 -1630.687,E2 -1630.687} C_VEL
LIN {X 0,Y 587.425,Z 526.568,A -85,B 0,C 180,E1 -1631.735,E2 -1631.735} C_VEL
LIN {X 0,Y 587.544,Z 515.85,A -85,B 0,C 180,E1 -1632.784,E2 -1632.784} C_VEL
LIN {X 0,Y 587.658,Z 502.977,A -85,B 0,C 180,E1 -1633.838,E2 -1633.838} C_VEL
LIN {X 0,Y 587.829,Z 489.954,A -85,B 0,C 180,E1 -1634.717,E2 -1634.717} C_VEL
LIN {X 0,Y 587.892,Z 479.431,A -85,B 0,C 180,E1 -1635.315,E2 -1635.315} C_VEL
LIN {X 0,Y 587.351,Z 474.26,A -85,B 0,C 180,E1 -1635.591,E2 -1635.591} C_VEL
LIN {X 0,Y 582.41,Z 459.109,A -85,B 0,C 180,E1 -1636.38,E2 -1636.38} C_VEL
LIN {X 0,Y 581.406,Z 453.742,A -85,B 0,C 180,E1 -1636.599,E2 -1636.599} C_VEL
LIN {X 0,Y 581.35,Z 451.895,A -85,B 0,C 180,E1 -1636.664,E2 -1636.664} C_VEL
LIN {X 0,Y 581.444,Z 436.687,A -85,B 0,C 180,E1 -1637.081,E2 -1637.081} C_VEL
LIN {X 0,Y 581.526,Z 421.525,A -85,B 0,C 180,E1 -1637.354,E2 -1637.354} C_VEL
LIN {X 0,Y 581.828,Z 268.981,A -85,B 0,C 180,E1 -1639.29,E2 -1639.29} C_VEL
LIN {X 0,Y 580.661,Z 263.436,A -85,B 0,C 180,E1 -1639.412,E2 -1639.412} C_VEL
LIN {X 0,Y 580.741,Z 253.546,A -85,B 0,C 180,E1 -1640.876,E2 -1640.876} C_VEL
LIN {X 0,Y 580.287,Z 250.828,A -85,B 0,C 180,E1 -1641.305,E2 -1641.305} C_VEL
LIN {X 0,Y 580.281,Z 250.827,A -85,B 0,C 180,E1 -1644.316,E2 -1644.316} C_VEL
LIN {X 0,Y 580.278,Z 250.825,A -85,B 0,C 180,E1 -1647.401,E2 -1647.401} C_VEL
LIN {X 0,Y 580.268,Z 250.832,A -85,B 0,C 180,E1 -1649.773,E2 -1649.773} C_VEL
LIN {X 0,Y 580.293,Z 250.825,A -85,B 0,C 180,E1 -1652.2,E2 -1652.2} C_VEL
LIN {X 0,Y 580.284,Z 250.822,A -85,B 0,C 180,E1 -1654.696,E2 -1654.696} C_VEL
LIN {X 0,Y 580.287,Z 250.823,A -85,B 0,C 180,E1 -1657.268,E2 -1657.268} C_VEL
LIN {X 0,Y 580.286,Z 250.825,A -85,B 0,C 180,E1 -1660.269,E2 -1660.269} C_VEL
LIN {X 0,Y 580.27,Z 250.823,A -85,B 0,C 180,E1 -1662.706,E2 -1662.706} C_VEL
LIN {X 0,Y 580.26,Z 250.831,A -85,B 0,C 180,E1 -1665.609,E2 -1665.609} C_VEL
LIN {X 0,Y 580.286,Z 250.825,A -85,B 0,C 180,E1 -1668.231,E2 -1668.231} C_VEL
LIN {X 0,Y 580.272,Z 250.823,A -85,B 0,C 180,E1 -1670.964,E2 -1670.964} C_VEL
LIN {X 0,Y 580.265,Z 250.831,A -85,B 0,C 180,E1 -1673.595,E2 -1673.595} C_VEL
LIN {X 0,Y 580.3,Z 250.823,A -85,B 0,C 180,E1 -1676.143,E2 -1676.143} C_VEL
LIN {X 0,Y 580.271,Z 250.823,A -85,B 0,C 180,E1 -1678.613,E2 -1678.613} C_VEL
LIN {X 0,Y 580.288,Z 250.822,A -85,B 0,C 180,E1 -1681.023,E2 -1681.023} C_VEL
LIN {X 0,Y 580.268,Z 250.827,A -85,B 0,C 180,E1 -1684.149,E2 -1684.149} C_VEL
LIN {X 0,Y 580.265,Z 250.824,A -85,B 0,C 180,E1 -1686.441,E2 -1686.441} C_VEL
LIN {X 0,Y 580.269,Z 250.829,A -85,B 0,C 180,E1 -1689.436,E2 -1689.436} C_VEL
LIN {X 0,Y 580.259,Z 250.835,A -85,B 0,C 180,E1 -1691.644,E2 -1691.644} C_VEL
LIN {X 0,Y 580.272,Z 250.83,A -85,B 0,C 180,E1 -1693.825,E2 -1693.825} C_VEL
LIN {X 0,Y 580.309,Z 250.823,A -85,B 0,C 180,E1 -1695.982,E2 -1695.982} C_VEL
LIN {X 0,Y 580.298,Z 250.82,A -85,B 0,C 180,E1 -1698.826,E2 -1698.826} C_VEL
LIN {X 0,Y 580.323,Z 250.826,A -85,B 0,C 180,E1 -1701.643,E2 -1701.643} C_VEL
LIN {X 0,Y 580.307,Z 250.818,A -85,B 0,C 180,E1 -1704.439,E2 -1704.439} C_VEL
LIN {X 0,Y 580.338,Z 250.819,A -85,B 0,C 180,E1 -1707.223,E2 -1707.223} C_VEL
LIN {X 0,Y 580.332,Z 250.819,A -85,B 0,C 180,E1 -1709.999,E2 -1709.999} C_VEL
LIN {X 0,Y 580.327,Z 250.816,A -85,B 0,C 180,E1 -1712.776,E2 -1712.776} C_VEL
LIN {X 0,Y 580.316,Z 250.827,A -85,B 0,C 180,E1 -1715.559,E2 -1715.559} C_VEL
LIN {X 0,Y 580.299,Z 250.82,A -85,B 0,C 180,E1 -1718.355,E2 -1718.355} C_VEL
LIN {X 0,Y 580.289,Z 250.826,A -85,B 0,C 180,E1 -1721.19,E2 -1721.19} C_VEL
LIN {X 0,Y 580.307,Z 250.821,A -85,B 0,C 180,E1 -1724.016,E2 -1724.016} C_VEL
LIN {X 0,Y 580.3,Z 250.821,A -85,B 0,C 180,E1 -1726.913,E2 -1726.913} C_VEL
LIN {X 0,Y 580.292,Z 250.824,A -85,B 0,C 180,E1 -1729.822,E2 -1729.822} C_VEL
LIN {X 0,Y 580.283,Z 250.823,A -85,B 0,C 180,E1 -1732.802,E2 -1732.802} C_VEL
LIN {X 0,Y 580.294,Z 250.825,A -85,B 0,C 180,E1 -1735.079,E2 -1735.079} C_VEL
LIN {X 0,Y 580.285,Z 250.822,A -85,B 0,C 180,E1 -1738.185,E2 -1738.185} C_VEL
LIN {X 0,Y 580.279,Z 250.823,A -85,B 0,C 180,E1 -1740.696,E2 -1740.696} C_VEL
LIN {X 0,Y 580.29,Z 250.83,A -85,B 0,C 180,E1 -1743.316,E2 -1743.316} C_VEL
LIN {X 0,Y 580.258,Z 250.828,A -85,B 0,C 180,E1 -1745.76,E2 -1745.76} C_VEL
LIN {X 0,Y 580.273,Z 250.823,A -85,B 0,C 180,E1 -1748.146,E2 -1748.146} C_VEL
LIN {X 0,Y 580.287,Z 250.824,A -85,B 0,C 180,E1 -1750.843,E2 -1750.843} C_VEL
LIN {X 0,Y 580.273,Z 250.827,A -85,B 0,C 180,E1 -1753.657,E2 -1753.657} C_VEL
LIN {X 0,Y 580.271,Z 250.824,A -85,B 0,C 180,E1 -1756.608,E2 -1756.608} C_VEL
LIN {X 0,Y 580.286,Z 250.83,A -85,B 0,C 180,E1 -1759.157,E2 -1759.157} C_VEL
LIN {X 0,Y 580.274,Z 250.824,A -85,B 0,C 180,E1 -1761.927,E2 -1761.927} C_VEL
LIN {X 0,Y 580.284,Z 250.822,A -85,B 0,C 180,E1 -1764.456,E2 -1764.456} C_VEL
LIN {X 0,Y 580.277,Z 250.828,A -85,B 0,C 180,E1 -1766.975,E2 -1766.975} C_VEL
LIN {X 0,Y 580.288,Z 250.827,A -85,B 0,C 180,E1 -1769.426,E2 -1769.426} C_VEL
LIN {X 0,Y 580.282,Z 250.821,A -85,B 0,C 180,E1 -1772.141,E2 -1772.141} C_VEL
LIN {X 0,Y 580.306,Z 250.827,A -85,B 0,C 180,E1 -1775.27,E2 -1775.27} C_VEL
LIN {X 0,Y 580.258,Z 250.825,A -85,B 0,C 180,E1 -1777.948,E2 -1777.948} C_VEL
LIN {X 0,Y 580.304,Z 250.825,A -85,B 0,C 180,E1 -1780.914,E2 -1780.914} C_VEL
LIN {X 0,Y 580.261,Z 250.825,A -85,B 0,C 180,E1 -1783.826,E2 -1783.826} C_VEL
LIN {X 0,Y 580.305,Z 250.819,A -85,B 0,C 180,E1 -1785.983,E2 -1785.983} C_VEL
LIN {X 0,Y 580.29,Z 250.826,A -85,B 0,C 180,E1 -1788.827,E2 -1788.827} C_VEL
LIN {X 0,Y 580.296,Z 250.822,A -85,B 0,C 180,E1 -1791.644,E2 -1791.644} C_VEL
LIN {X 0,Y 580.314,Z 250.819,A -85,B 0,C 180,E1 -1794.441,E2 -1794.441} C_VEL
LIN {X 0,Y 580.326,Z 250.823,A -85,B 0,C 180,E1 -1797.224,E2 -1797.224} C_VEL
LIN {X 0,Y 580.328,Z 250.816,A -85,B 0,C 180,E1 -1800.001,E2 -1800.001} C_VEL
LIN {X 0,Y 580.338,Z 250.821,A -85,B 0,C 180,E1 -1802.777,E2 -1802.777} C_VEL
LIN {X 0,Y 580.304,Z 250.821,A -85,B 0,C 180,E1 -1805.56,E2 -1805.56} C_VEL
LIN {X 0,Y 580.319,Z 250.818,A -85,B 0,C 180,E1 -1808.357,E2 -1808.357} C_VEL
LIN {X 0,Y 580.322,Z 250.822,A -85,B 0,C 180,E1 -1811.209,E2 -1811.209} C_VEL
LIN {X 0,Y 580.302,Z 250.821,A -85,B 0,C 180,E1 -1814.339,E2 -1814.339} C_VEL
LIN {X 0,Y 580.303,Z 250.83,A -85,B 0,C 180,E1 -1816.915,E2 -1816.915} C_VEL
LIN {X 0,Y 580.277,Z 250.822,A -85,B 0,C 180,E1 -1819.824,E2 -1819.824} C_VEL
LIN {X 0,Y 580.269,Z 250.823,A -85,B 0,C 180,E1 -1822.053,E2 -1822.053} C_VEL
LIN {X 0,Y 580.29,Z 250.827,A -85,B 0,C 180,E1 -1825.081,E2 -1825.081} C_VEL
LIN {X 0,Y 580.289,Z 250.822,A -85,B 0,C 180,E1 -1828.186,E2 -1828.186} C_VEL
LIN {X 0,Y 580.274,Z 250.83,A -85,B 0,C 180,E1 -1830.696,E2 -1830.696} C_VEL
LIN {X 0,Y 580.274,Z 250.825,A -85,B 0,C 180,E1 -1833.314,E2 -1833.314} C_VEL
LIN {X 0,Y 580.237,Z 250.827,A -85,B 0,C 180,E1 -1835.758,E2 -1835.758} C_VEL
LIN {X 0,Y 580.278,Z 250.823,A -85,B 0,C 180,E1 -1838.147,E2 -1838.147} C_VEL
LIN {X 0,Y 580.287,Z 250.83,A -85,B 0,C 180,E1 -1840.845,E2 -1840.845} C_VEL
LIN {X 0,Y 580.261,Z 250.824,A -85,B 0,C 180,E1 -1843.66,E2 -1843.66} C_VEL
LIN {X 0,Y 580.268,Z 250.831,A -85,B 0,C 180,E1 -1846.611,E2 -1846.611} C_VEL
LIN {X 0,Y 580.29,Z 250.824,A -85,B 0,C 180,E1 -1849.158,E2 -1849.158} C_VEL
LIN {X 0,Y 580.28,Z 250.823,A -85,B 0,C 180,E1 -1851.929,E2 -1851.929} C_VEL
LIN {X 0,Y 580.244,Z 250.833,A -85,B 0,C 180,E1 -1854.454,E2 -1854.454} C_VEL
LIN {X 0,Y 580.282,Z 250.827,A -85,B 0,C 180,E1 -1856.976,E2 -1856.976} C_VEL
LIN {X 0,Y 580.283,Z 250.824,A -85,B 0,C 180,E1 -1859.426,E2 -1859.426} C_VEL
LIN {X 0,Y 580.283,Z 250.827,A -85,B 0,C 180,E1 -1862.144,E2 -1862.144} C_VEL
LIN {X 0,Y 580.318,Z 250.908,A -85,B 0,C 180,E1 -1862.628,E2 -1862.628} C_VEL
LIN {X 0,Y 581.682,Z 257.521,A -85,B 0,C 180,E1 -1863.447,E2 -1863.447} C_VEL
LIN {X 0,Y 581.444,Z 280.945,A -85,B 0,C 180,E1 -1866.115,E2 -1866.115} C_VEL
LIN {X 0,Y 581.098,Z 307.601,A -85,B 0,C 180,E1 -1869.098,E2 -1869.098} C_VEL
LIN {X 0,Y 580.943,Z 321.411,A -85,B 0,C 180,E1 -1870.623,E2 -1870.623} C_VEL
LIN {X 0,Y 581.901,Z 326.661,A -85,B 0,C 180,E1 -1870.728,E2 -1870.728} C_VEL
LIN {X 0,Y 581.523,Z 488.044,A -85,B 0,C 180,E1 -1872.789,E2 -1872.789} C_VEL
LIN {X 0,Y 581.426,Z 503.749,A -85,B 0,C 180,E1 -1873.137,E2 -1873.137} C_VEL
LIN {X 0,Y 581.246,Z 519.072,A -85,B 0,C 180,E1 -1873.629,E2 -1873.629} C_VEL
LIN {X 0,Y 581.123,Z 532.794,A -85,B 0,C 180,E1 -1874.211,E2 -1874.211} C_VEL
LIN {X 0,Y 580.942,Z 546.262,A -85,B 0,C 180,E1 -1874.925,E2 -1874.925} C_VEL
LIN {X 0,Y 580.802,Z 559.496,A -85,B 0,C 180,E1 -1875.784,E2 -1875.784} C_VEL
LIN {X 0,Y 580.608,Z 571.302,A -85,B 0,C 180,E1 -1876.705,E2 -1876.705} C_VEL
LIN {X 0,Y 580.478,Z 582.76,A -85,B 0,C 180,E1 -1877.769,E2 -1877.769} C_VEL
LIN {X 0,Y 580.307,Z 593.456,A -85,B 0,C 180,E1 -1878.954,E2 -1878.954} C_VEL
LIN {X 0,Y 580.268,Z 601.865,A -85,B 0,C 180,E1 -1880.063,E2 -1880.063} C_VEL
LIN {X 0,Y 580.213,Z 609.739,A -85,B 0,C 180,E1 -1881.292,E2 -1881.292} C_VEL
LIN {X 0,Y 580.13,Z 617.094,A -85,B 0,C 180,E1 -1882.693,E2 -1882.693} C_VEL
LIN {X 0,Y 580.129,Z 622.927,A -85,B 0,C 180,E1 -1884.091,E2 -1884.091} C_VEL
LIN {X 0,Y 580.041,Z 626.388,A -85,B 0,C 180,E1 -1885.136,E2 -1885.136} C_VEL
LIN {X 0,Y 580.104,Z 629.891,A -85,B 0,C 180,E1 -1886.528,E2 -1886.528} C_VEL
LIN {X 0,Y 580.037,Z 632.194,A -85,B 0,C 180,E1 -1887.918,E2 -1887.918} C_VEL
LIN {X 0,Y 580.038,Z 633.35,A -85,B 0,C 180,E1 -1889.307,E2 -1889.307} C_VEL
LIN {X 0,Y 580.038,Z 633.349,A -85,B 0,C 180,E1 -1890.695,E2 -1890.695} C_VEL
LIN {X 0,Y 580.037,Z 632.19,A -85,B 0,C 180,E1 -1892.084,E2 -1892.084} C_VEL
LIN {X 0,Y 580.105,Z 629.885,A -85,B 0,C 180,E1 -1893.474,E2 -1893.474} C_VEL
LIN {X 0,Y 580.041,Z 626.382,A -85,B 0,C 180,E1 -1894.866,E2 -1894.866} C_VEL
LIN {X 0,Y 580.091,Z 621.605,A -85,B 0,C 180,E1 -1896.261,E2 -1896.261} C_VEL
LIN {X 0,Y 580.166,Z 615.419,A -85,B 0,C 180,E1 -1897.658,E2 -1897.658} C_VEL
LIN {X 0,Y 580.208,Z 607.644,A -85,B 0,C 180,E1 -1899.061,E2 -1899.061} C_VEL
LIN {X 0,Y 580.309,Z 599.363,A -85,B 0,C 180,E1 -1900.291,E2 -1900.291} C_VEL
LIN {X 0,Y 580.384,Z 589.387,A -85,B 0,C 180,E1 -1901.526,E2 -1901.526} C_VEL
LIN {X 0,Y 580.542,Z 579.181,A -85,B 0,C 180,E1 -1902.587,E2 -1902.587} C_VEL
LIN {X 0,Y 580.689,Z 567.008,A -85,B 0,C 180,E1 -1903.652,E2 -1903.652} C_VEL
LIN {X 0,Y 580.849,Z 554.792,A -85,B 0,C 180,E1 -1904.542,E2 -1904.542} C_VEL
LIN {X 0,Y 581.007,Z 541.503,A -85,B 0,C 180,E1 -1905.344,E2 -1905.344} C_VEL
LIN {X 0,Y 581.2,Z 526.816,A -85,B 0,C 180,E1 -1906.059,E2 -1906.059} C_VEL
LIN {X 0,Y 581.343,Z 512.592,A -85,B 0,C 180,E1 -1906.596,E2 -1906.596} C_VEL
LIN {X 0,Y 581.456,Z 498.131,A -85,B 0,C 180,E1 -1907.002,E2 -1907.002} C_VEL
LIN {X 0,Y 581.523,Z 483.76,A -85,B 0,C 180,E1 -1907.276,E2 -1907.276} C_VEL
LIN {X 0,Y 581.835,Z 326.145,A -85,B 0,C 180,E1 -1909.281,E2 -1909.281} C_VEL
LIN {X 0,Y 580.944,Z 321.266,A -85,B 0,C 180,E1 -1909.393,E2 -1909.393} C_VEL
LIN {X 0,Y 581.224,Z 295.921,A -85,B 0,C 180,E1 -1912.202,E2 -1912.202} C_VEL
LIN {X 0,Y 581.547,Z 270.93,A -85,B 0,C 180,E1 -1915.023,E2 -1915.023} C_VEL
LIN {X 0,Y 581.616,Z 257.054,A -85,B 0,C 180,E1 -1916.596,E2 -1916.596} C_VEL
LIN {X 0,Y 580.325,Z 250.827,A -85,B 0,C 180,E1 -1917.352,E2 -1917.352} C_VEL
LIN {X 0,Y 580.279,Z 250.826,A -85,B 0,C 180,E1 -1919.774,E2 -1919.774} C_VEL
LIN {X 0,Y 580.3,Z 250.822,A -85,B 0,C 180,E1 -1922.201,E2 -1922.201} C_VEL
LIN {X 0,Y 580.291,Z 250.826,A -85,B 0,C 180,E1 -1924.697,E2 -1924.697} C_VEL
LIN {X 0,Y 580.302,Z 250.827,A -85,B 0,C 180,E1 -1927.269,E2 -1927.269} C_VEL
LIN {X 0,Y 580.299,Z 250.822,A -85,B 0,C 180,E1 -1930.271,E2 -1930.271} C_VEL
LIN {X 0,Y 580.281,Z 250.83,A -85,B 0,C 180,E1 -1932.707,E2 -1932.707} C_VEL
LIN {X 0,Y 580.273,Z 250.824,A -85,B 0,C 180,E1 -1935.61,E2 -1935.61} C_VEL
LIN {X 0,Y 580.286,Z 250.825,A -85,B 0,C 180,E1 -1938.231,E2 -1938.231} C_VEL
LIN {X 0,Y 580.277,Z 250.828,A -85,B 0,C 180,E1 -1940.965,E2 -1940.965} C_VEL
LIN {X 0,Y 580.254,Z 250.826,A -85,B 0,C 180,E1 -1943.595,E2 -1943.595} C_VEL
LIN {X 0,Y 580.319,Z 250.823,A -85,B 0,C 180,E1 -1946.145,E2 -1946.145} C_VEL
LIN {X 0,Y 580.28,Z 250.83,A -85,B 0,C 180,E1 -1948.614,E2 -1948.614} C_VEL
LIN {X 0,Y 580.293,Z 250.823,A -85,B 0,C 180,E1 -1951.024,E2 -1951.024} C_VEL
LIN {X 0,Y 580.286,Z 250.831,A -85,B 0,C 180,E1 -1954.15,E2 -1954.15} C_VEL
LIN {X 0,Y 580.275,Z 250.832,A -85,B 0,C 180,E1 -1956.442,E2 -1956.442} C_VEL
LIN {X 0,Y 580.309,Z 250.85,A -85,B 0,C 180,E1 -1958.795,E2 -1958.795} C_VEL
LIN {X 0,Y 580.788,Z 255.16,A -85,B 0,C 180,E1 -1959.456,E2 -1959.456} C_VEL
LIN {X 0,Y 580.69,Z 263.745,A -85,B 0,C 180,E1 -1960.694,E2 -1960.694} C_VEL
LIN {X 0,Y 581.91,Z 269.498,A -85,B 0,C 180,E1 -1960.809,E2 -1960.809} C_VEL
LIN {X 0,Y 581.518,Z 428.172,A -85,B 0,C 180,E1 -1962.839,E2 -1962.839} C_VEL
LIN {X 0,Y 581.404,Z 443.605,A -85,B 0,C 180,E1 -1963.18,E2 -1963.18} C_VEL
LIN {X 0,Y 581.255,Z 457.721,A -85,B 0,C 180,E1 -1963.628,E2 -1963.628} C_VEL
LIN {X 0,Y 581.137,Z 471.808,A -85,B 0,C 180,E1 -1964.21,E2 -1964.21} C_VEL
LIN {X 0,Y 580.947,Z 485.405,A -85,B 0,C 180,E1 -1964.924,E2 -1964.924} C_VEL
LIN {X 0,Y 580.811,Z 498.893,A -85,B 0,C 180,E1 -1965.786,E2 -1965.786} C_VEL
LIN {X 0,Y 580.611,Z 510.722,A -85,B 0,C 180,E1 -1966.703,E2 -1966.703} C_VEL
LIN {X 0,Y 580.484,Z 522.315,A -85,B 0,C 180,E1 -1967.767,E2 -1967.767} C_VEL
LIN {X 0,Y 580.323,Z 532.996,A -85,B 0,C 180,E1 -1968.946,E2 -1968.946} C_VEL
LIN {X 0,Y 580.271,Z 541.549,A -85,B 0,C 180,E1 -1970.061,E2 -1970.061} C_VEL
LIN {X 0,Y 580.181,Z 550.478,A -85,B 0,C 180,E1 -1971.466,E2 -1971.466} C_VEL
LIN {X 0,Y 580.134,Z 556.892,A -85,B 0,C 180,E1 -1972.692,E2 -1972.692} C_VEL
LIN {X 0,Y 580.129,Z 562.761,A -85,B 0,C 180,E1 -1974.089,E2 -1974.089} C_VEL
LIN {X 0,Y 580.039,Z 566.258,A -85,B 0,C 180,E1 -1975.134,E2 -1975.134} C_VEL
LIN {X 0,Y 580.107,Z 569.793,A -85,B 0,C 180,E1 -1976.527,E2 -1976.527} C_VEL
LIN {X 0,Y 580.034,Z 572.15,A -85,B 0,C 180,E1 -1977.916,E2 -1977.916} C_VEL
LIN {X 0,Y 580.037,Z 573.318,A -85,B 0,C 180,E1 -1979.305,E2 -1979.305} C_VEL
LIN {X 0,Y 580.039,Z 573.346,A -85,B 0,C 180,E1 -1980.694,E2 -1980.694} C_VEL
LIN {X 0,Y 580.037,Z 572.254,A -85,B 0,C 180,E1 -1982.083,E2 -1982.083} C_VEL
LIN {X 0,Y 580.108,Z 569.983,A -85,B 0,C 180,E1 -1983.472,E2 -1983.472} C_VEL
LIN {X 0,Y 580.042,Z 566.533,A -85,B 0,C 180,E1 -1984.865,E2 -1984.865} C_VEL
LIN {X 0,Y 580.096,Z 561.794,A -85,B 0,C 180,E1 -1986.259,E2 -1986.259} C_VEL
LIN {X 0,Y 580.138,Z 555.634,A -85,B 0,C 180,E1 -1987.657,E2 -1987.657} C_VEL
LIN {X 0,Y 580.207,Z 547.945,A -85,B 0,C 180,E1 -1989.059,E2 -1989.059} C_VEL
LIN {X 0,Y 580.288,Z 539.67,A -85,B 0,C 180,E1 -1990.29,E2 -1990.29} C_VEL
LIN {X 0,Y 580.38,Z 529.794,A -85,B 0,C 180,E1 -1991.524,E2 -1991.524} C_VEL
LIN {X 0,Y 580.513,Z 519.634,A -85,B 0,C 180,E1 -1992.586,E2 -1992.586} C_VEL
LIN {X 0,Y 580.652,Z 508.62,A -85,B 0,C 180,E1 -1993.562,E2 -1993.562} C_VEL
LIN {X 0,Y 580.841,Z 495.51,A -85,B 0,C 180,E1 -1994.538,E2 -1994.538} C_VEL
LIN {X 0,Y 580.974,Z 482.301,A -85,B 0,C 180,E1 -1995.344,E2 -1995.344} C_VEL
LIN {X 0,Y 581.178,Z 467.852,A -85,B 0,C 180,E1 -1996.058,E2 -1996.058} C_VEL
LIN {X 0,Y 581.322,Z 453.904,A -85,B 0,C 180,E1 -1996.595,E2 -1996.595} C_VEL
LIN {X 0,Y 581.35,Z 451.895,A -85,B 0,C 180,E1 -1996.664,E2 -1996.664} C_VEL
LIN {X 0,Y 580.751,Z 448.202,A -85,B 0,C 180,E1 -1996.803,E2 -1996.803} C_VEL
LIN {X 0,Y 575.307,Z 436.74,A -85,B 0,C 180,E1 -1997.267,E2 -1997.267} C_VEL
LIN {X 0,Y 574.721,Z 432.945,A -85,B 0,C 180,E1 -1997.369,E2 -1997.369} C_VEL
LIN {X 0,Y 574.766,Z 413.008,A -85,B 0,C 180,E1 -1997.676,E2 -1997.676} C_VEL
LIN {X 0,Y 575.14,Z 270.063,A -85,B 0,C 180,E1 -1999.509,E2 -1999.509} C_VEL
LIN {X 0,Y 573.726,Z 263.407,A -85,B 0,C 180,E1 -1999.66,E2 -1999.66} C_VEL
LIN {X 0,Y 573.69,Z 254.104,A -85,B 0,C 180,E1 -2001.06,E2 -2001.06} C_VEL
LIN {X 0,Y 573.256,Z 251.704,A -85,B 0,C 180,E1 -2001.442,E2 -2001.442} C_VEL
LIN {X 0,Y 573.216,Z 251.712,A -85,B 0,C 180,E1 -2003.865,E2 -2003.865} C_VEL
LIN {X 0,Y 573.215,Z 251.705,A -85,B 0,C 180,E1 -2006.487,E2 -2006.487} C_VEL
LIN {X 0,Y 573.229,Z 251.702,A -85,B 0,C 180,E1 -2008.564,E2 -2008.564} C_VEL
LIN {X 0,Y 573.219,Z 251.702,A -85,B 0,C 180,E1 -2010.993,E2 -2010.993} C_VEL
LIN {X 0,Y 573.262,Z 251.7,A -85,B 0,C 180,E1 -2013.523,E2 -2013.523} C_VEL
LIN {X 0,Y 573.192,Z 251.712,A -85,B 0,C 180,E1 -2016.052,E2 -2016.052} C_VEL
LIN {X 0,Y 573.236,Z 251.699,A -85,B 0,C 180,E1 -2018.701,E2 -2018.701} C_VEL
LIN {X 0,Y 573.223,Z 251.707,A -85,B 0,C 180,E1 -2021.591,E2 -2021.591} C_VEL
LIN {X 0,Y 573.226,Z 251.703,A -85,B 0,C 180,E1 -2024.333,E2 -2024.333} C_VEL
LIN {X 0,Y 573.234,Z 251.703,A -85,B 0,C 180,E1 -2027.358,E2 -2027.358} C_VEL
LIN {X 0,Y 573.234,Z 251.701,A -85,B 0,C 180,E1 -2030.391,E2 -2030.391} C_VEL
LIN {X 0,Y 573.248,Z 251.699,A -85,B 0,C 180,E1 -2033.076,E2 -2033.076} C_VEL
LIN {X 0,Y 573.262,Z 251.705,A -85,B 0,C 180,E1 -2035.67,E2 -2035.67} C_VEL
LIN {X 0,Y 573.236,Z 251.703,A -85,B 0,C 180,E1 -2038.183,E2 -2038.183} C_VEL
LIN {X 0,Y 573.258,Z 251.697,A -85,B 0,C 180,E1 -2040.633,E2 -2040.633} C_VEL
LIN {X 0,Y 573.226,Z 251.707,A -85,B 0,C 180,E1 -2043.507,E2 -2043.507} C_VEL
LIN {X 0,Y 573.22,Z 251.705,A -85,B 0,C 180,E1 -2046.133,E2 -2046.133} C_VEL
LIN {X 0,Y 573.245,Z 251.701,A -85,B 0,C 180,E1 -2049.173,E2 -2049.173} C_VEL
LIN {X 0,Y 573.215,Z 251.708,A -85,B 0,C 180,E1 -2051.41,E2 -2051.41} C_VEL
LIN {X 0,Y 573.25,Z 251.707,A -85,B 0,C 180,E1 -2053.621,E2 -2053.621} C_VEL
LIN {X 0,Y 573.258,Z 251.704,A -85,B 0,C 180,E1 -2055.806,E2 -2055.806} C_VEL
LIN {X 0,Y 573.256,Z 251.697,A -85,B 0,C 180,E1 -2058.744,E2 -2058.744} C_VEL
LIN {X 0,Y 573.279,Z 251.703,A -85,B 0,C 180,E1 -2061.54,E2 -2061.54} C_VEL
LIN {X 0,Y 573.275,Z 251.695,A -85,B 0,C 180,E1 -2064.371,E2 -2064.371} C_VEL
LIN {X 0,Y 573.292,Z 251.697,A -85,B 0,C 180,E1 -2067.891,E2 -2067.891} C_VEL
LIN {X 0,Y 573.32,Z 251.689,A -85,B 0,C 180,E1 -2070.701,E2 -2070.701} C_VEL
LIN {X 0,Y 573.233,Z 251.71,A -85,B 0,C 180,E1 -2073.514,E2 -2073.514} C_VEL
LIN {X 0,Y 573.282,Z 251.702,A -85,B 0,C 180,E1 -2075.627,E2 -2075.627} C_VEL
LIN {X 0,Y 573.265,Z 251.702,A -85,B 0,C 180,E1 -2077.749,E2 -2077.749} C_VEL
LIN {X 0,Y 573.253,Z 251.697,A -85,B 0,C 180,E1 -2080.596,E2 -2080.596} C_VEL
LIN {X 0,Y 573.252,Z 251.698,A -85,B 0,C 180,E1 -2082.748,E2 -2082.748} C_VEL
LIN {X 0,Y 573.224,Z 251.703,A -85,B 0,C 180,E1 -2084.919,E2 -2084.919} C_VEL
LIN {X 0,Y 573.23,Z 251.704,A -85,B 0,C 180,E1 -2087.848,E2 -2087.848} C_VEL
LIN {X 0,Y 573.239,Z 251.7,A -85,B 0,C 180,E1 -2090.076,E2 -2090.076} C_VEL
LIN {X 0,Y 573.221,Z 251.706,A -85,B 0,C 180,E1 -2093.099,E2 -2093.099} C_VEL
LIN {X 0,Y 573.241,Z 251.709,A -85,B 0,C 180,E1 -2095.409,E2 -2095.409} C_VEL
LIN {X 0,Y 573.237,Z 251.7,A -85,B 0,C 180,E1 -2098.028,E2 -2098.028} C_VEL
LIN {X 0,Y 573.225,Z 251.703,A -85,B 0,C 180,E1 -2100.883,E2 -2100.883} C_VEL
LIN {X 0,Y 573.248,Z 251.705,A -85,B 0,C 180,E1 -2103.523,E2 -2103.523} C_VEL
LIN {X 0,Y 573.227,Z 251.701,A -85,B 0,C 180,E1 -2106.049,E2 -2106.049} C_VEL
LIN {X 0,Y 573.234,Z 251.701,A -85,B 0,C 180,E1 -2108.7,E2 -2108.7} C_VEL
LIN {X 0,Y 573.217,Z 251.709,A -85,B 0,C 180,E1 -2111.456,E2 -2111.456} C_VEL
LIN {X 0,Y 573.224,Z 251.701,A -85,B 0,C 180,E1 -2114.333,E2 -2114.333} C_VEL
LIN {X 0,Y 573.229,Z 251.709,A -85,B 0,C 180,E1 -2117.358,E2 -2117.358} C_VEL
LIN {X 0,Y 573.232,Z 251.7,A -85,B 0,C 180,E1 -2120.393,E2 -2120.393} C_VEL
LIN {X 0,Y 573.238,Z 251.707,A -85,B 0,C 180,E1 -2123.078,E2 -2123.078} C_VEL
LIN {X 0,Y 573.259,Z 251.7,A -85,B 0,C 180,E1 -2125.672,E2 -2125.672} C_VEL
LIN {X 0,Y 573.233,Z 251.7,A -85,B 0,C 180,E1 -2128.185,E2 -2128.185} C_VEL
LIN {X 0,Y 573.249,Z 251.7,A -85,B 0,C 180,E1 -2130.634,E2 -2130.634} C_VEL
LIN {X 0,Y 573.223,Z 251.706,A -85,B 0,C 180,E1 -2133.507,E2 -2133.507} C_VEL
LIN {X 0,Y 573.215,Z 251.702,A -85,B 0,C 180,E1 -2136.135,E2 -2136.135} C_VEL
LIN {X 0,Y 573.246,Z 251.708,A -85,B 0,C 180,E1 -2139.174,E2 -2139.174} C_VEL
LIN {X 0,Y 573.211,Z 251.708,A -85,B 0,C 180,E1 -2141.412,E2 -2141.412} C_VEL
LIN {X 0,Y 573.234,Z 251.702,A -85,B 0,C 180,E1 -2143.622,E2 -2143.622} C_VEL
LIN {X 0,Y 573.252,Z 251.698,A -85,B 0,C 180,E1 -2145.807,E2 -2145.807} C_VEL
LIN {X 0,Y 573.248,Z 251.702,A -85,B 0,C 180,E1 -2148.745,E2 -2148.745} C_VEL
LIN {X 0,Y 573.241,Z 251.702,A -85,B 0,C 180,E1 -2151.541,E2 -2151.541} C_VEL
LIN {X 0,Y 573.221,Z 251.703,A -85,B 0,C 180,E1 -2153.665,E2 -2153.665} C_VEL
LIN {X 0,Y 573.201,Z 251.704,A -85,B 0,C 180,E1 -2155.782,E2 -2155.782} C_VEL
LIN {X 0,Y 573.286,Z 251.693,A -85,B 0,C 180,E1 -2157.893,E2 -2157.893} C_VEL
LIN {X 0,Y 573.329,Z 251.693,A -85,B 0,C 180,E1 -2160.703,E2 -2160.703} C_VEL
LIN {X 0,Y 573.218,Z 251.704,A -85,B 0,C 180,E1 -2163.515,E2 -2163.515} C_VEL
LIN {X 0,Y 573.271,Z 251.696,A -85,B 0,C 180,E1 -2165.629,E2 -2165.629} C_VEL
LIN {X 0,Y 573.276,Z 251.697,A -85,B 0,C 180,E1 -2168.46,E2 -2168.46} C_VEL
LIN {X 0,Y 573.267,Z 251.7,A -85,B 0,C 180,E1 -2171.313,E2 -2171.313} C_VEL
LIN {X 0,Y 573.268,Z 251.698,A -85,B 0,C 180,E1 -2174.425,E2 -2174.425} C_VEL
LIN {X 0,Y 573.247,Z 251.705,A -85,B 0,C 180,E1 -2177.112,E2 -2177.112} C_VEL
LIN {X 0,Y 573.235,Z 251.7,A -85,B 0,C 180,E1 -2180.078,E2 -2180.078} C_VEL
LIN {X 0,Y 573.234,Z 251.702,A -85,B 0,C 180,E1 -2182.338,E2 -2182.338} C_VEL
LIN {X 0,Y 573.234,Z 251.702,A -85,B 0,C 180,E1 -2185.411,E2 -2185.411} C_VEL
LIN {X 0,Y 573.239,Z 251.699,A -85,B 0,C 180,E1 -2188.03,E2 -2188.03} C_VEL
LIN {X 0,Y 573.235,Z 251.701,A -85,B 0,C 180,E1 -2190.177,E2 -2190.177} C_VEL
LIN {X 0,Y 573.244,Z 251.705,A -85,B 0,C 180,E1 -2192.646,E2 -2192.646} C_VEL
LIN {X 0,Y 573.199,Z 251.708,A -85,B 0,C 180,E1 -2195.189,E2 -2195.189} C_VEL
LIN {X 0,Y 573.225,Z 251.701,A -85,B 0,C 180,E1 -2197.809,E2 -2197.809} C_VEL
LIN {X 0,Y 573.235,Z 251.705,A -85,B 0,C 180,E1 -2200.526,E2 -2200.526} C_VEL
LIN {X 0,Y 573.223,Z 251.702,A -85,B 0,C 180,E1 -2203.361,E2 -2203.361} C_VEL
LIN {X 0,Y 573.237,Z 251.703,A -85,B 0,C 180,E1 -2206.332,E2 -2206.332} C_VEL
LIN {X 0,Y 573.22,Z 251.708,A -85,B 0,C 180,E1 -2208.544,E2 -2208.544} C_VEL
LIN {X 0,Y 573.237,Z 251.701,A -85,B 0,C 180,E1 -2211.3,E2 -2211.3} C_VEL
LIN {X 0,Y 573.187,Z 251.707,A -85,B 0,C 180,E1 -2214.022,E2 -2214.022} C_VEL
LIN {X 0,Y 573.264,Z 251.703,A -85,B 0,C 180,E1 -2216.519,E2 -2216.519} C_VEL
LIN {X 0,Y 573.222,Z 251.706,A -85,B 0,C 180,E1 -2219.119,E2 -2219.119} C_VEL
LIN {X 0,Y 573.237,Z 251.704,A -85,B 0,C 180,E1 -2221.974,E2 -2221.974} C_VEL
LIN {X 0,Y 573.274,Z 251.86,A -85,B 0,C 180,E1 -2222.409,E2 -2222.409} C_VEL
LIN {X 0,Y 574.903,Z 259.403,A -85,B 0,C 180,E1 -2223.359,E2 -2223.359} C_VEL
LIN {X 0,Y 574.634,Z 282.611,A -85,B 0,C 180,E1 -2226.006,E2 -2226.006} C_VEL
LIN {X 0,Y 574.237,Z 309.319,A -85,B 0,C 180,E1 -2229.03,E2 -2229.03} C_VEL
LIN {X 0,Y 574.041,Z 321.389,A -85,B 0,C 180,E1 -2230.378,E2 -2230.378} C_VEL
LIN {X 0,Y 575.22,Z 328.666,A -85,B 0,C 180,E1 -2230.521,E2 -2230.521} C_VEL
LIN {X 0,Y 574.751,Z 488.267,A -85,B 0,C 180,E1 -2232.584,E2 -2232.584} C_VEL
LIN {X 0,Y 574.62,Z 503.747,A -85,B 0,C 180,E1 -2232.931,E2 -2232.931} C_VEL
LIN {X 0,Y 574.403,Z 519.07,A -85,B 0,C 180,E1 -2233.428,E2 -2233.428} C_VEL
LIN {X 0,Y 574.291,Z 532.797,A -85,B 0,C 180,E1 -2234.018,E2 -2234.018} C_VEL
LIN {X 0,Y 574.047,Z 546.264,A -85,B 0,C 180,E1 -2234.74,E2 -2234.74} C_VEL
LIN {X 0,Y 573.858,Z 559.835,A -85,B 0,C 180,E1 -2235.633,E2 -2235.633} C_VEL
LIN {X 0,Y 573.635,Z 572.363,A -85,B 0,C 180,E1 -2236.63,E2 -2236.63} C_VEL
LIN {X 0,Y 573.476,Z 582.76,A -85,B 0,C 180,E1 -2237.617,E2 -2237.617} C_VEL
LIN {X 0,Y 573.285,Z 592.778,A -85,B 0,C 180,E1 -2238.735,E2 -2238.735} C_VEL
LIN {X 0,Y 573.242,Z 601.865,A -85,B 0,C 180,E1 -2239.94,E2 -2239.94} C_VEL
LIN {X 0,Y 573.132,Z 609.74,A -85,B 0,C 180,E1 -2241.184,E2 -2241.184} C_VEL
LIN {X 0,Y 573.074,Z 617.094,A -85,B 0,C 180,E1 -2242.603,E2 -2242.603} C_VEL
LIN {X 0,Y 573.039,Z 622.927,A -85,B 0,C 180,E1 -2244.017,E2 -2244.017} C_VEL
LIN {X 0,Y 572.951,Z 626.388,A -85,B 0,C 180,E1 -2245.075,E2 -2245.075} C_VEL
LIN {X 0,Y 573.004,Z 629.891,A -85,B 0,C 180,E1 -2246.485,E2 -2246.485} C_VEL
LIN {X 0,Y 572.937,Z 632.193,A -85,B 0,C 180,E1 -2247.892,E2 -2247.892} C_VEL
LIN {X 0,Y 572.938,Z 633.349,A -85,B 0,C 180,E1 -2249.298,E2 -2249.298} C_VEL
LIN {X 0,Y 572.938,Z 633.349,A -85,B 0,C 180,E1 -2250.704,E2 -2250.704} C_VEL
LIN {X 0,Y 572.937,Z 632.189,A -85,B 0,C 180,E1 -2252.11,E2 -2252.11} C_VEL
LIN {X 0,Y 573.004,Z 629.885,A -85,B 0,C 180,E1 -2253.517,E2 -2253.517} C_VEL
LIN {X 0,Y 572.951,Z 626.383,A -85,B 0,C 180,E1 -2254.927,E2 -2254.927} C_VEL
LIN {X 0,Y 573.012,Z 621.605,A -85,B 0,C 180,E1 -2256.338,E2 -2256.338} C_VEL
LIN {X 0,Y 573.094,Z 615.418,A -85,B 0,C 180,E1 -2257.753,E2 -2257.753} C_VEL
LIN {X 0,Y 573.137,Z 607.643,A -85,B 0,C 180,E1 -2259.174,E2 -2259.174} C_VEL
LIN {X 0,Y 573.271,Z 599.362,A -85,B 0,C 180,E1 -2260.419,E2 -2260.419} C_VEL
LIN {X 0,Y 573.387,Z 589.384,A -85,B 0,C 180,E1 -2261.669,E2 -2261.669} C_VEL
LIN {X 0,Y 573.569,Z 579.18,A -85,B 0,C 180,E1 -2262.743,E2 -2262.743} C_VEL
LIN {X 0,Y 573.743,Z 567.009,A -85,B 0,C 180,E1 -2263.82,E2 -2263.82} C_VEL
LIN {X 0,Y 573.964,Z 553.891,A -85,B 0,C 180,E1 -2264.782,E2 -2264.782} C_VEL
LIN {X 0,Y 574.114,Z 541.5,A -85,B 0,C 180,E1 -2265.533,E2 -2265.533} C_VEL
LIN {X 0,Y 574.338,Z 526.813,A -85,B 0,C 180,E1 -2266.256,E2 -2266.256} C_VEL
LIN {X 0,Y 574.544,Z 512.592,A -85,B 0,C 180,E1 -2266.798,E2 -2266.798} C_VEL
LIN {X 0,Y 574.704,Z 497.556,A -85,B 0,C 180,E1 -2267.223,E2 -2267.223} C_VEL
LIN {X 0,Y 574.757,Z 482.624,A -85,B 0,C 180,E1 -2267.503,E2 -2267.503} C_VEL
LIN {X 0,Y 575.154,Z 327.241,A -85,B 0,C 180,E1 -2269.5,E2 -2269.5} C_VEL
LIN {X 0,Y 574.056,Z 321.319,A -85,B 0,C 180,E1 -2269.63,E2 -2269.63} C_VEL
LIN {X 0,Y 574.387,Z 297.587,A -85,B 0,C 180,E1 -2272.291,E2 -2272.291} C_VEL
LIN {X 0,Y 574.717,Z 273.163,A -85,B 0,C 180,E1 -2275.062,E2 -2275.062} C_VEL
LIN {X 0,Y 574.679,Z 257.882,A -85,B 0,C 180,E1 -2276.779,E2 -2276.779} C_VEL
LIN {X 0,Y 573.256,Z 251.706,A -85,B 0,C 180,E1 -2277.569,E2 -2277.569} C_VEL
LIN {X 0,Y 573.24,Z 251.701,A -85,B 0,C 180,E1 -2280.177,E2 -2280.177} C_VEL
LIN {X 0,Y 573.255,Z 251.702,A -85,B 0,C 180,E1 -2282.646,E2 -2282.646} C_VEL
LIN {X 0,Y 573.21,Z 251.713,A -85,B 0,C 180,E1 -2285.188,E2 -2285.188} C_VEL
LIN {X 0,Y 573.238,Z 251.701,A -85,B 0,C 180,E1 -2287.808,E2 -2287.808} C_VEL
LIN {X 0,Y 573.25,Z 251.703,A -85,B 0,C 180,E1 -2290.525,E2 -2290.525} C_VEL
LIN {X 0,Y 573.241,Z 251.703,A -85,B 0,C 180,E1 -2293.36,E2 -2293.36} C_VEL
LIN {X 0,Y 573.25,Z 251.702,A -85,B 0,C 180,E1 -2296.331,E2 -2296.331} C_VEL
LIN {X 0,Y 573.235,Z 251.708,A -85,B 0,C 180,E1 -2298.543,E2 -2298.543} C_VEL
LIN {X 0,Y 573.243,Z 251.701,A -85,B 0,C 180,E1 -2301.298,E2 -2301.298} C_VEL
LIN {X 0,Y 573.198,Z 251.708,A -85,B 0,C 180,E1 -2304.021,E2 -2304.021} C_VEL
LIN {X 0,Y 573.275,Z 251.705,A -85,B 0,C 180,E1 -2306.518,E2 -2306.518} C_VEL
